//取收集瓶暂存工位到仓库
		80:
			ParameterList3:=2;            //取2号大夹持工具
			A00_取放工具();
			IF 取工具完成 THEN
				取工具完成:=FALSE;
				机器人流程:=81;
			END_IF
		81:
			A71_取暂存收集瓶放仓库();
			IF 取暂存收集瓶组放仓库完成 THEN
				collect_Old_Plate_Slot:=0;
				FunctionID:=0;
				机器人流程:=0;
				取暂存收集瓶组放仓库完成:=FALSE;
			END_IF		
		
		
		
		
		
	
	
	


//取收集器暂存工位到仓库
		90:
			ParameterList3:=2;            //取2号大夹持工具
			A00_取放工具();
			IF 取工具完成 THEN
				取工具完成:=FALSE;
				机器人流程:=91;
			END_IF
		91:
			A70_取暂存收集器组放仓库();
			IF 取暂存收集器组放仓库完成 THEN
				scrape_Old_Plate_Slot:=0;
				FunctionID:=0;
				机器人流程:=0;
				取暂存收集器组放仓库完成:=FALSE;
			END_IF	







//取暂存收集器到刮取位
		100:
			ParameterList3:=3;                           //取3号小夹持工具
			A00_取放工具();
			IF 取工具完成 THEN
				取工具完成:=FALSE;
				机器人流程:=101;
			END_IF	
		101:
			A45_取暂存收集器放刮板位();
			IF 取暂存收集器放刮板位完成 THEN
				scrape_Consume_Slot:=0;
				FunctionID:=0;
				取暂存收集器放刮板位完成:=FALSE;
				机器人流程:=0;
			END_IF
			
			






//取刮板拍照收集器到收集工位
		110:
			ParameterList3:=3;                           //取3号小夹持工具
			A00_取放工具();
			IF 取工具完成 THEN
				取工具完成:=FALSE;
				机器人流程:=111;
			END_IF
		111:
			A55_取刮板收集器放到收集工位();
			IF 取刮板收集器放到收集工位完成 THEN
				FunctionID:=0;
				取刮板收集器放到收集工位完成:=FALSE;
				机器人流程:=0;
			END_IF
			
	
	
	
	
	
	
	
//取暂存收集瓶到收集工位	
		120:
			ParameterList3:=3;                           //取3号小夹持工具
			A00_取放工具();
			IF 取工具完成 THEN
				取工具完成:=FALSE;
				机器人流程:=121;
			END_IF
		121:
			A50_取暂存收集瓶放收集工位();
			IF 取暂存收集瓶放收集工位完成 THEN
				FunctionID:=0;
				取暂存收集瓶放收集工位完成:=FALSE;
				机器人流程:=0;
			END_IF
			
			






//取收集器到暂存工位
		130:
			ParameterList3:=3;                           //取3号小夹持工具
			A00_取放工具();
			IF 取工具完成 THEN
				取工具完成:=FALSE;
				机器人流程:=131;
			END_IF
		131:
			A60_取收集器放暂存工位();
			IF 取收集器放暂存工位完成 THEN
				collect_Powder_Return_Slot:=0;
				收集器组站位符:=FALSE;
				收集工位放收集器完成:=TRUE;
				FunctionID:=0;
				机器人流程:=0;
				取收集器放暂存工位完成:=FALSE;
			END_IF
			
			




//取收集瓶到暂存工位
		140:
			ParameterList3:=3;                           //取3号小夹持工具
			A00_取放工具();
			IF 取工具完成 THEN
				取工具完成:=FALSE;
				机器人流程:=141;
			END_IF
		141:
			A65_取收集瓶放暂存工位();
			IF 取收集瓶放暂存工位完成 THEN
				scrape_Consume_Slot:=0;
				收集瓶组站位符:=FALSE;
				FunctionID:=0;
				机器人流程:=0;
				取收集瓶放暂存工位完成:=FALSE;
			END_IF
			


    END_CASE
END_IF

ACTION A55_取刮板收集器放到收集工位:



CASE 取刮板收集器放到收集工位step OF
	0:
		地轨轴11YDATE.fAbsTarget:=HMI_地轨轴11Y.position[2];     //地轨去取收集组位置暂存位置
			地轨轴11YDATE.xMoveAbs:=TRUE;
			取刮板收集器放到收集工位step:=1;
	1:
		IF 地轨轴11YDATE.bAbMoveDone AND 拍照工位允许取收集器 AND  Status=0 THEN
			地轨轴11YDATE.xMoveAbs:=FALSE;
			拍照工位机器人退出工位完成:=FALSE;
			FunctionID:=11;
			Execute:=1;
			ParameterList5:=4;                          //机器人去夹持工位
			取刮板收集器放到收集工位step:=10;
		END_IF
	10:
		IF RO_ParameterList5=4 THEN
			拍照工位机器人到达收集器夹持位:=TRUE;
			取刮板收集器放到收集工位step:=20;
		END_IF
	20:
		IF 拍照工位机器人退出 THEN
			
			拍照工位机器人到达收集器夹持位:=FALSE;
			ParameterList5:=5;                          //机器人退出工位
			取刮板收集器放到收集工位step:=30;
		END_IF
	30:
		IF RO_ParameterList5=5 THEN
			拍照工位机器人退出完成:=TRUE;
			Execute:=0;
			地轨轴11YDATE.fAbsTarget:=HMI_地轨轴11Y.position[3];     //地轨去收集工位
			地轨轴11YDATE.xMoveAbs:=TRUE;
			取刮板收集器放到收集工位step:=40;
		END_IF
	40:
		IF 地轨轴11YDATE.bAbMoveDone THEN
			地轨轴11YDATE.xMoveAbs:=FALSE;                     
			取刮板收集器放到收集工位step:=50;
		END_IF
	50:
		IF 收集工位允许放收集器 AND  Status=0 THEN
			FunctionID:=12;                             //放收集工位收集器
			ParameterList8:=1;                         //机器人放收集器到夹持工位
			Execute:=1;
			取刮板收集器放到收集工位step:=60;
		END_IF
	60:
		IF RO_ParameterList8=1 THEN
			
			收集工位放收集器到工位:=TRUE;
			取刮板收集器放到收集工位step:=70;
		END_IF
	70:
		IF 收集工位允许机器人退出工位 THEN
			ParameterList8:=2;                     //机器人退出工位
			取刮板收集器放到收集工位step:=80;
		END_IF
	80:
		IF RO_ParameterList8=2 AND Status=2 THEN                //机器人退出工位完成
			Execute:=0;
			收集工位机器人退出完成:=TRUE;
			收集工位放收集器到工位:=FALSE;
			取刮板收集器放到收集工位完成:=TRUE;
			取刮板收集器放到收集工位step:=0;
		END_IF
END_CASE
END_ACTION

ACTION A00_取放工具:



CASE 取工具setp OF
	0:
		IF RO_ParameterList3=ParameterList3 THEN
			取工具完成:=TRUE;
			取工具setp:=0;
		ELSE
			取工具setp:=5;
		END_IF
	5:
		地轨轴11YDATE.fAbsTarget:=HMI_地轨轴11Y.position[4];     //地轨去取工具位置
		地轨轴11YDATE.xMoveAbs:=TRUE;
		IF 地轨轴11YDATE.bAbMoveDone THEN
			地轨轴11YDATE.xMoveAbs:=FALSE;
			FunctionID:=23;                              //取工具ID
			Execute:=1;                                  //机器人启动                        
			取工具setp:=10;
		END_IF
	10:
		IF RO_ParameterList3=ParameterList3 AND Status=2 THEN                               //取工具完成                                   
			Execute:=0;
			取工具完成:=TRUE;
			取工具setp:=0;
		END_IF
END_CASE
END_ACTION

ACTION A15_放点样硅胶板:



CASE 放点样硅胶板step OF
	0:	IF  Status=0 THEN
	  		ParameterList4:=0;
			FunctionID:=2;                         //放点样硅胶板
			ParameterList2:=1;                     //机器人放硅胶板
			Execute:=1;
			放点样硅胶板step:=10;
	  	END_IF
		
	10:
		IF RO_ParameterList2=1 AND Status=2 THEN         //机器人放硅胶板完成
			上样点样放硅胶板完成:=TRUE;
			Execute:=0;
			放点样硅胶板完成:=TRUE;
			放点样硅胶板step:=0;
		END_IF
END_CASE
END_ACTION

ACTION A65_取收集瓶放暂存工位:

CASE 取收集瓶放暂存工位step OF
	0:
		地轨轴11YDATE.fAbsTarget:=HMI_地轨轴11Y.position[3];     //地轨去取收集组位置暂存位置
			地轨轴11YDATE.xMoveAbs:=TRUE;
			取收集瓶放暂存工位step:=5;
	5:
		IF 地轨轴11YDATE.bAbMoveDone AND 收集工位允许机器人取收集瓶放暂存工位 THEN
			地轨轴11YDATE.xMoveAbs:=FALSE;
			收集工位放收集瓶完成:=FALSE;
			FunctionID:=12;
			ParameterList8:=4;                               //到收集工位取收集瓶
			Execute:=1;
			取收集瓶放暂存工位step:=6;
		END_IF
	6:
		
		IF  RO_ParameterList8=4 AND Status=2 THEN
			取收集瓶放暂存工位step:=10;
			收集工位机器人放收集瓶到暂存工位完成:=TRUE;
			Execute:=0;
		END_IF
	10:
		IF Status=0 THEN
			ParameterList8:=5;                               //放收集瓶到暂存工位
			Execute:=1;
			ParameterList9:=collect_Consume_Slot;
			取收集瓶放暂存工位step:=20;
		END_IF
	20:
		IF RO_ParameterList8=5 AND Status=2 THEN                         //放收集瓶到暂存工位完成
			Execute:=0;
			取收集瓶放暂存工位step:=0;
			取收集瓶放暂存工位完成:=TRUE;
		END_IF
END_CASE
END_ACTION

ACTION A71_取暂存收集瓶放仓库:






CASE 取暂存收集瓶组放仓库step OF
	0:
		地轨轴11YDATE.fAbsTarget:=HMI_地轨轴11Y.position[3];     //地轨去取收集组位置暂存位置
		地轨轴11YDATE.xMoveAbs:=TRUE;
		溶液收集瓶定位自动:=FALSE;
		取暂存收集瓶组放仓库step:=10;
	10:
		IF 地轨轴11YDATE.bAbMoveDone AND  Status=0 THEN
			地轨轴11YDATE.xMoveAbs:=FALSE;
			FunctionID:=14;                              //放收集器/瓶到仓库
			ParameterList6:=16;                          //取暂存收集器组
			Execute:=1; 
			取暂存收集瓶组放仓库step:=20;
		END_IF
	20:
		IF RO_ParameterList6=16 AND Status=2 THEN                      //取完成
			Execute:=0; 
			地轨轴11YDATE.fAbsTarget:=HMI_地轨轴11Y.position[6];     //地轨去放收集组位置
			地轨轴11YDATE.xMoveAbs:=TRUE;
			取暂存收集瓶组放仓库step:=30;
		END_IF
	30:
		IF 地轨轴11YDATE.bAbMoveDone AND Status=0 THEN
			地轨轴11YDATE.xMoveAbs:=FALSE;
			ParameterList6:=collect_Old_Plate_Slot+6;               //取暂存收集瓶组
			Execute:=1; 
			取暂存收集瓶组放仓库step:=40;
		END_IF
	40:
		IF RO_ParameterList6=collect_Old_Plate_Slot+6  AND Status=2 THEN
			取暂存收集瓶组放仓库完成:=TRUE;
			Execute:=0; 
			取暂存收集瓶组放仓库step:=0;
		END_IF
END_CASE
END_ACTION

ACTION A20_取点样硅胶板:



CASE 取点样硅胶板step OF
	0:
		地轨轴11YDATE.fAbsTarget:=HMI_地轨轴11Y.position[1];     //地轨去上样点样位置
			地轨轴11YDATE.xMoveAbs:=TRUE;
			IF 地轨轴11YDATE.bAbMoveDone THEN
				地轨轴11YDATE.xMoveAbs:=FALSE; 
				取点样硅胶板step:=5;
			END_IF
	5:
		IF  Status=0 THEN    //上样点样完成，展开准备完成
			FunctionID:=3;                              //取点样硅胶板
			ParameterList2:=2;                          //取硅胶板参数
			Execute:=1;                                  //机器人启动                        
			取点样硅胶板step:=10;
		END_IF
	10:
		IF RO_ParameterList2=2 AND Status=2 THEN
			Execute:=0;
			ParameterList2:=0;
			上样点样允许取硅胶板:=FALSE;
			取点样硅胶板完成:=TRUE;
			取点样硅胶板step:=0;
		END_IF
END_CASE
END_ACTION

ACTION A60_取收集器放暂存工位:


CASE 取收集器放暂存工位step OF
	0:
		地轨轴11YDATE.fAbsTarget:=HMI_地轨轴11Y.position[3];     //地轨去取收集组位置暂存位置
			地轨轴11YDATE.xMoveAbs:=TRUE;
			取收集器放暂存工位step:=5;
			
	5:
		IF 地轨轴11YDATE.bAbMoveDone  THEN
			地轨轴11YDATE.xMoveAbs:=FALSE;
			FunctionID:=12;  
			ParameterList8:=6;                               //放收集器回暂存工位
			Execute:=1;
			取收集器放暂存工位step:=10;
		END_IF
	10:
		IF RO_ParameterList8=6  THEN                       //放收集器回暂存工位完成
			收集工位机器人到达收集器位置:=TRUE;
			取收集器放暂存工位step:=30;
		END_IF
	30:
		IF 收集工位机器人取收集器放回暂存工位 THEN
			ParameterList8:=7;                               //机器人去取收集器
			ParameterList7:=collect_Powder_Return_Slot;
			收集工位机器人取收集器放回暂存工位:=FALSE;
			取收集器放暂存工位step:=40;
		END_IF
	40:
		IF RO_ParameterList8=7 AND Status=2 THEN                         //到达夹持位置
			Execute:=0;
			取收集器放暂存工位完成:=TRUE;
			取收集器放暂存工位step:=0;
		END_IF
END_CASE
END_ACTION

ACTION A10_取升降机硅胶板:


CASE 取升降硅胶板step OF
		0:
			地轨轴11YDATE.fAbsTarget:=HMI_地轨轴11Y.position[1];     //地轨去上样点样位置
			地轨轴11YDATE.xMoveAbs:=TRUE;
			IF 地轨轴11YDATE.bAbMoveDone THEN
				地轨轴11YDATE.xMoveAbs:=FALSE; 
				IF 升降上料伺服允许取料 AND Status=0 THEN
					FunctionID:=1;                              //取升降硅胶板ID
					ParameterList4:=1;                           //去升降机构位置
					Execute:=1;                                  //机器人启动 
					取升降硅胶板step:=10;
				END_IF
			END_IF
			
		10:
			IF RO_ParameterList4=1 THEN                   //机器人到位
				升降上料机器人已吸住物料:=TRUE;
				取升降硅胶板step:=15;
			END_IF
		15:
			IF 升降上料伺服下降完成  THEN
				ParameterList4:=2;                        //机器人取物料
				取升降硅胶板step:=20;
			END_IF
			
		20:
			IF RO_ParameterList4=2 AND Status=2 THEN                //机器人取物料完成
				ParameterList4:=0;
				Execute:=0;
				升降上料机器人取料完成:=TRUE;
				取升降硅胶板完成:=TRUE;
				取升降硅胶板step:=0;
			END_IF
END_CASE
END_ACTION

ACTION A25_放展缸硅胶板:



CASE 放展缸硅胶板step OF
	0:	
		地轨轴11YDATE.fAbsTarget:=HMI_地轨轴11Y.position[5];     //地轨去展开位
		地轨轴11YDATE.xMoveAbs:=TRUE;
		IF 地轨轴11YDATE.bAbMoveDone AND Status=0 THEN
			地轨轴11YDATE.xMoveAbs:=FALSE;
			展开工位机器人到达准备点:=TRUE;
			放展缸硅胶板step:=5;
		END_IF
	5:
		IF 展开工位允许放硅胶板 THEN
			FunctionID:=4;                              //放展缸硅胶板
			Execute:=1;                                  //机器人启动       
			展开工位机器人到达准备点:=FALSE;
			放展缸硅胶板step:=10;
		END_IF
			
	10:
		IF RO_ParameterList1>0 AND Status=2 THEN                       //放硅胶板完成
			展开工位机器人放硅胶板完成:=TRUE;
			FunctionID:=0;
			Execute:=0;
			放展缸硅胶板step:=0;
		END_IF
END_CASE
END_ACTION

ACTION A41_取收集瓶组放暂存工位:


CASE 取收集瓶组放暂存工位step OF
	0:
			地轨轴11YDATE.fAbsTarget:=HMI_地轨轴11Y.position[6];     //地轨去取收集组位置
			地轨轴11YDATE.xMoveAbs:=TRUE;
			溶液收集瓶定位自动:=FALSE;
			取收集瓶组放暂存工位step:=10;
	10:
		IF 地轨轴11YDATE.bAbMoveDone AND Status=0 THEN
				地轨轴11YDATE.xMoveAbs:=FALSE;
				FunctionID:=21;                              //取收集瓶组
				ParameterList6:=collect_Fetch_Rack_Plate+6;       //取收集瓶组坐标
				Execute:=1;                                  //机器人启动                        
				取收集瓶组放暂存工位step:=20;
			END_IF
	20:
		IF RO_ParameterList6=ParameterList6 AND Status=2 THEN             //取收集瓶组完成
			Execute:=0;
			地轨轴11YDATE.fAbsTarget:=HMI_地轨轴11Y.position[3];     //地轨去收集工位
			地轨轴11YDATE.xMoveAbs:=TRUE;
			取收集瓶组放暂存工位step:=30;
		END_IF
	30:
		IF 地轨轴11YDATE.bAbMoveDone AND Status=0 THEN
				地轨轴11YDATE.xMoveAbs:=FALSE;
				FunctionID:=22;                              //放收集瓶组
				ParameterList6:=14;                         //放收集瓶组
				Execute:=1;                                  //机器人启动                        
				取收集瓶组放暂存工位step:=40;
		END_IF
	40:
		IF RO_ParameterList6=14 AND Status=2 THEN                        //放收集瓶完成
			Execute:=0; 
			ParameterList6:=0;
			溶液收集瓶定位自动:=TRUE;
			取收集瓶组放暂存工位完成:=TRUE;
			取收集瓶组放暂存工位step:=0;
		END_IF
END_CASE
END_ACTION

ACTION A65_放废料硅胶板:



CASE 取刮板硅胶板放废料区step OF
	0:
		地轨轴11YDATE.fAbsTarget:=HMI_地轨轴11Y.position[1];     //地轨去上样点样位置
			地轨轴11YDATE.xMoveAbs:=TRUE;
			IF 地轨轴11YDATE.bAbMoveDone THEN
				地轨轴11YDATE.xMoveAbs:=FALSE;
				取刮板硅胶板放废料区step:=5;
            END_IF
	5:
		IF  升降下料伺服允许放料 AND  Status=0 THEN
			
			FunctionID:=8; 
			ParameterList4:=3;                                     //机器人放到废料区
			Execute:=1; 
			取刮板硅胶板放废料区step:=10;
		END_IF
	10:
		IF RO_ParameterList4=3 AND Status=2  THEN                               //机器人放废料区完成
			Execute:=0; 
			刮板拍照工位站位符:=FALSE;
			升降下料机器人放废料完成:=TRUE;
			取刮板硅胶板放废料区完成:=TRUE;
			取刮板硅胶板放废料区step:=0;
		END_IF
END_CASE
END_ACTION

ACTION A35_放拍照硅胶板:




CASE 放拍照硅胶板step OF
	0:
		地轨轴11YDATE.fAbsTarget:=HMI_地轨轴11Y.position[2];     //地轨去刮板拍照位
		地轨轴11YDATE.xMoveAbs:=TRUE;
		IF 地轨轴11YDATE.bAbMoveDone AND Status=0 THEN
				地轨轴11YDATE.xMoveAbs:=FALSE;
				FunctionID:=6;                              //放拍照硅胶板
				ParameterList5:=1;                           //放硅胶板到刮板拍照位
				Execute:=1;                                  //机器人启动                        
				放拍照硅胶板step:=10;
		END_IF
	10:
		IF RO_ParameterList5=1 AND Status=2 THEN              //放硅胶板完成
			Execute:=0; 
			ParameterList5:=0;
			拍照工位放硅胶板完成:=TRUE;
			放拍照硅胶板完成:=TRUE;
			放拍照硅胶板step:=0;
		END_IF
END_CASE
END_ACTION

ACTION A45_取暂存收集器放刮板位:


CASE 取暂存收集器放刮板位step OF
	0:
		IF RO_ParameterList3=3 THEN
			ParameterList3:=0;
			Execute:=0;
			地轨轴11YDATE.fAbsTarget:=HMI_地轨轴11Y.position[2];     //地轨去刮板拍照位
			地轨轴11YDATE.xMoveAbs:=TRUE;
			取暂存收集器放刮板位step:=10;
		END_IF
	10:
		IF 地轨轴11YDATE.bAbMoveDone THEN
			地轨轴11YDATE.xMoveAbs:=FALSE;                     
			取暂存收集器放刮板位step:=20;
		END_IF
	20:
		IF 拍照工位允许放收集器 AND Status=0 THEN
			FunctionID:=9;                              //取暂存收集器
			ParameterList7:=scrape_Consume_Slot;           //取收集器
			Execute:=1;
			取暂存收集器放刮板位step:=30;
		END_IF
	30:
		IF RO_ParameterList7=ParameterList7  THEN                   //取收集器完成
			Execute:=0;
			取暂存收集器放刮板位step:=40;
		END_IF
	40:
		IF Status=0 THEN
			FunctionID:=10;                             //放收集器
			ParameterList5:=2;                         //机器人放收集器到夹持工位
			Execute:=1;
			取暂存收集器放刮板位step:=45;
		END_IF
	45:
		IF RO_ParameterList5=2 THEN
			拍照工位机器人到达夹持位:=TRUE;
			取暂存收集器放刮板位step:=50;
		END_IF
	50:
		IF 拍照工位机器人退出工位 THEN
			ParameterList5:=3;                         //机器人退出工位
			拍照工位机器人到达夹持位:=FALSE;
			取暂存收集器放刮板位step:=60;
		END_IF
	60:
		IF RO_ParameterList5=3 AND Status=2 THEN                    //机器人退出工位完成
			Execute:=0;
			拍照工位机器人退出工位完成:=TRUE;
			取暂存收集器放刮板位完成:=TRUE;
			取暂存收集器放刮板位step:=0;
		END_IF	
	
	
	
	
END_CASE
END_ACTION

ACTION A40_取收集器组放暂存工位:




CASE 取收集器组放暂存工位step OF
	0:
		地轨轴11YDATE.fAbsTarget:=HMI_地轨轴11Y.position[6];     //地轨去取收集组位置
		地轨轴11YDATE.xMoveAbs:=TRUE;
		取收集器组放暂存工位step:=10;
	
	10:
		IF 地轨轴11YDATE.bAbMoveDone  AND Status=0 THEN
				地轨轴11YDATE.xMoveAbs:=FALSE;
				FunctionID:=19;                              //取收集器组
				ParameterList6:=scrape_Fetch_Rack_Plate;       //取收集器组坐标
				Execute:=1;                                  //机器人启动                        
				取收集器组放暂存工位step:=20;
			END_IF
	20:
		IF RO_ParameterList6=ParameterList6 AND Status=2 THEN             //取收集器组完成
			Execute:=0;
			地轨轴11YDATE.fAbsTarget:=HMI_地轨轴11Y.position[3];     //地轨去收集
			地轨轴11YDATE.xMoveAbs:=TRUE;
			取收集器组放暂存工位step:=30;
		END_IF
	30:
		IF 地轨轴11YDATE.bAbMoveDone AND Status=0 THEN
				地轨轴11YDATE.xMoveAbs:=FALSE;
				FunctionID:=20;                              //放收集器组
				ParameterList6:=13;                         //取收集器组坐标
				Execute:=1;                                  //机器人启动                        
				取收集器组放暂存工位step:=40;
		END_IF
	40:
		IF RO_ParameterList6=13  AND Status=2 THEN                        //放收集器完成
			Execute:=0; 
			粉末收集器定位自动:=TRUE;
			取收集器组放暂存工位完成:=TRUE;
			取收集器组放暂存工位step:=0;
		END_IF
	
END_CASE
END_ACTION

ACTION A50_取暂存收集瓶放收集工位:




CASE 取暂存收集瓶放收集工位step OF
	0:
		地轨轴11YDATE.fAbsTarget:=HMI_地轨轴11Y.position[3];     //地轨去取收集组位置暂存位置
			地轨轴11YDATE.xMoveAbs:=TRUE;
			取暂存收集瓶放收集工位step:=1;
	1:
		IF 地轨轴11YDATE.bAbMoveDone AND Status=0 THEN
			地轨轴11YDATE.xMoveAbs:=FALSE;
			FunctionID:=13;                             //取收集瓶
			ParameterList9:=collect_Consume_Slot;           //取收集瓶参数
			Execute:=1;
			取暂存收集瓶放收集工位step:=5;
		END_IF
	5:
		IF RO_ParameterList9=ParameterList9 AND 收集工位允许放收集瓶 THEN        //取收集瓶完成
			Execute:=0;
			取暂存收集瓶放收集工位step:=6;
		END_IF
	6:
		IF Status=0 THEN
			FunctionID:=15;  
			ParameterList8:=3;
			Execute:=1;
			取暂存收集瓶放收集工位step:=10;
		END_IF
	10:
		IF RO_ParameterList8=3 AND Status=2 THEN
				Execute:=0;
			收集工位放收集瓶完成:=TRUE;
			取暂存收集瓶放收集工位完成:=TRUE;
			取暂存收集瓶放收集工位step:=0;
		END_IF
END_CASE
END_ACTION

ACTION A70_取暂存收集器组放仓库:


CASE 取暂存收集器组放仓库step OF
	0:
		IF RO_ParameterList3=2 THEN
			Execute:=0; 
			地轨轴11YDATE.fAbsTarget:=HMI_地轨轴11Y.position[3];     //地轨去取收集组位置暂存位置
			地轨轴11YDATE.xMoveAbs:=TRUE;
			取暂存收集器组放仓库step:=10;
			粉末收集器定位自动:=FALSE;
		END_IF
	10:
		IF 地轨轴11YDATE.bAbMoveDone AND  Status=0 THEN
			地轨轴11YDATE.xMoveAbs:=FALSE;
			粉末收集器定位自动:=FALSE;
			溶液收集瓶定位自动:=FALSE;
			FunctionID:=14;                              //放收集器/瓶到仓库
			ParameterList6:=15;                          //取暂存收集器组
			Execute:=1; 
			取暂存收集器组放仓库step:=20;
		END_IF
	20:
		IF RO_ParameterList6=15 AND  Status=2 THEN                      //取完成
			Execute:=0; 
			地轨轴11YDATE.fAbsTarget:=HMI_地轨轴11Y.position[6];     //地轨去放收集组位置
			地轨轴11YDATE.xMoveAbs:=TRUE;
			取暂存收集器组放仓库step:=30;
		END_IF
	30:
		IF 地轨轴11YDATE.bAbMoveDone AND  Status=0 THEN
			地轨轴11YDATE.xMoveAbs:=FALSE;
			ParameterList6:=scrape_Old_Plate_Slot;               //取暂存收集器组
			Execute:=1;
			取暂存收集器组放仓库step:=40;
		END_IF
	40:
		IF RO_ParameterList6=scrape_Old_Plate_Slot AND Status=2 THEN
			Execute:=0;
			取暂存收集器组放仓库完成:=TRUE;
			取暂存收集器组放仓库step:=0;
		END_IF
	
END_CASE
END_ACTION

ACTION A30_取展缸硅胶板:




CASE 取展缸硅胶板step OF
	0:
		地轨轴11YDATE.fAbsTarget:=HMI_地轨轴11Y.position[5];     //地轨去展开位
		地轨轴11YDATE.xMoveAbs:=TRUE;
		IF 地轨轴11YDATE.bAbMoveDone THEN
			地轨轴11YDATE.xMoveAbs:=FALSE;
			取展缸硅胶板step:=10;
		END_IF
	10:
		IF  ParameterList1>0 AND Status=0 THEN
			FunctionID:=5;                                  //取展缸硅胶板
			Execute:=1;
			取展缸硅胶板step:=20;
		END_IF
	20:
		IF RO_ParameterList1>0 AND Status=2 THEN                       //取硅胶板完成
			Execute:=0;
			取展缸硅胶板完成:=TRUE;
			取展缸硅胶板step:=0;
		END_IF
END_CASE
END_ACTION

ACTION A32_取拍照硅胶板:
CASE 取拍照硅胶完step OF
	0:
		地轨轴11YDATE.fAbsTarget:=HMI_地轨轴11Y.position[2];     //地轨去刮板拍照位
		地轨轴11YDATE.xMoveAbs:=TRUE;
		IF 地轨轴11YDATE.bAbMoveDone THEN
				地轨轴11YDATE.xMoveAbs:=FALSE;
				取拍照硅胶完step:=5;
		END_IF
	5:		
		IF (拍照工位允许取硅胶板去展开 OR 拍照工位允许取硅胶板放废料区) AND Status=0 THEN    
			FunctionID:=6;                              
			ParameterList5:=6;                           //机器人取硅胶板
			Execute:=1;             
			拍照工位允许取硅胶板去展开 := FALSE;
			取拍照硅胶完step:=10;
		END_IF
	10:
		IF RO_ParameterList5=6 AND Status=2 THEN
			Execute:=0;
			ParameterList6:=0;
			取拍照硅胶板完成:=TRUE;
			取拍照硅胶完step:=0;
		IF 拍照工位允许取硅胶板放废料区 THEN
			拍照工位机器人取硅胶板完成 := TRUE;
		END_IF
		END_IF
END_CASE
END_ACTION

END_PROGRAM

// Device/Application/25_FB_功能块/FB_RB_Control
FUNCTION_BLOCK FB_RB_Control
VAR_INPUT
	StartCmd     : BOOL;
StopCmd      : BOOL;
PauseCmd     : BOOL;
Reset:BOOL;
RobotRunning : BOOL;
RobotStopped : BOOL;
RobotPaused  : BOOL;
RobotAlarm   : BOOL;
PowerOn:BOOL;
END_VAR
VAR_OUTPUT
	StartOut     : BOOL;
StopOut      : BOOL;
PauseOut     : BOOL;
ResetOut:BOOL;
StatusRun    : BOOL;
StatusStop   : BOOL;
StatusPause  : BOOL;
StatusAlarm  : BOOL;
PowerOnOut:BOOL;
END_VAR
VAR
	State        : INT := 0;   // 当前状态
END_VAR

(* ================= 报警优先 ================= *)
IF RobotAlarm THEN
    State := 4;
END_IF

CASE State OF

    (* -------- 0：空闲 -------- *)
    0:
        StartOut := FALSE;
        StopOut  := TRUE;
        PauseOut := FALSE;
		ResetOut:=FALSE;
        IF StartCmd AND NOT RobotAlarm THEN
            State := 1;
        END_IF

    (* -------- 1：运行 -------- *)
    1:
		IF NOT PowerOn THEN
			PowerOnOut:=TRUE;
		ELSE
			PowerOnOut:=FALSE;
		END_IF
		IF PowerOn THEN
			StartOut := TRUE;
			StopOut  := FALSE;
			PauseOut := FALSE;
		END_IF
        

        IF StopCmd THEN
            State := 3;
        ELSIF PauseCmd THEN
            State := 2;
        
        END_IF

    (* -------- 2：暂停 -------- *)
    2:
        PauseOut := TRUE;
		StartOut := FALSE ;
        StopOut  := FALSE;
        IF StopCmd THEN
            State := 3;
        ELSIF  StartCmd AND NOT RobotAlarm THEN
            State := 1;
        END_IF

    (* -------- 3：停止 -------- *)
    3:
        StartOut := FALSE;
        StopOut  := TRUE;
        PauseOut := FALSE;

        IF RobotStopped THEN
            State := 0;
        END_IF

    (* -------- 4：报警 -------- *)
    4:
        StartOut := FALSE;
        StopOut  := TRUE;
        PauseOut := FALSE;

        IF  Reset THEN
			ResetOut:=TRUE;
            State := 0;
        END_IF

END_CASE

(* ================= 状态输出 ================= *)
StatusRun   := (State = 1);
StatusPause := (State = 2);
StatusStop  := (State = 0) OR (State = 3);
StatusAlarm := (State = 4);

END_FUNCTION_BLOCK

// Device/Application/40_Man/Develop_TankDrain
PROGRAM Develop_TankDrain
VAR
	i           : INT;      // 循环索引
    anyDraining : BOOL;     // 全局真空泵控制标志
	// 全局真空泵控制标志
	展开step: INT;
	// 全局真空泵控制标志
	TON_3: TON;
	// 全局真空泵控制标志
	TON_4: TON;
	BlowTimer: ARRAY[1..8] OF TON;
	BlowDuration: TIME := t#30s;
END_VAR




A50_Expand_liquid_discharge_排液();

ACTION A50_Expand_liquid_discharge_排液:

// ══════════════════════════════════════════════════════════════
// 排液控制程序（per-tank 并行 FSM，每扫描周期调用）
// ══════════════════════════════════════════════════════════════
// 程序名：PRG_TankDrain
// 文件名：plc_develop_drain.txt
// 职责：监控 Tank_Drain_Enable[1..8]，触发对应缸的 3 阶段排液流程
// 触发条件：Tank_Drain_Enable[i]=TRUE 且 Tank_State[i]=40
// 完成标志：Tank_Drain_Done[i]=TRUE, Tank_State[i]=99
// 复位方式：PC 写 Tank_Drain_Enable[i]=FALSE → 清 Done；
//           PC 写 Tank_State[i]=0 → 释放缸
// ══════════════════════════════════════════════════════════════
// 3 阶段排液时序（工程师已验证）：
//   Phase A — Draining(50)：开排液阀 + 真空泵，等待 DrainDuration
//   Phase B — BlowAir(55) ：追加开吹气阀，等待 BlowDuration
//   Phase C — CylinderRetract(60)：关所有阀 + 气缸退回，等待到位传感器
// ══════════════════════════════════════════════════════════════
// 硬件拓扑：
//   - 每缸有独立排液电磁阀、吹气电磁阀、气缸（伸出/退回）
//   - 真空泵（大真空泵）全局共享，anyDraining 引用计数式控制
//   - 排液气泡传感器按组共享（仅用于监控，不参与控制逻辑）
//   - 支持 8 缸完全并行排液（各缸 FSM 独立推进）
// ══════════════════════════════════════════════════════════════
// Tank_State 状态转换（排液相关）：
//   40 (Developing)      → 50 (Draining)        : Drain_Enable[i] 触发
//   50 (Draining)        → 55 (BlowAir)         : DrainTimer[i].Q
//   55 (BlowAir)         → 60 (CylinderRetract) : BlowTimer[i].Q
//   60 (CylinderRetract) → 99 (Done)            : 气缸到位传感器
//   99 (Done)            → 0  (Idle)            : PC 写 Tank_State=0
//   50/55/60             → 90 (Error)           : 急停
//   注：55/60 为 PLC 内部子状态，PC 只关心 Drain_Done（state 99）
// ══════════════════════════════════════════════════════════════
// 物理 IO 映射表（工程师变量名 → 缸索引）：
//   i=1: 展缸1排液电池阀1自动 / 展缸1吹气电池阀1自动 / 展缸1气缸1自动 / 展缸1气缸1动点
//   i=2: 展缸1排液电池阀2自动 / 展缸1吹气电池阀2自动 / 展缸1气缸2自动 / 展缸1气缸2动点
//   i=3: 展缸1排液电池阀3自动 / 展缸1吹气电池阀3自动 / 展缸1气缸3自动 / 展缸1气缸3动点
//   i=4: 展缸1排液电池阀4自动 / 展缸1吹气电池阀4自动 / 展缸1气缸4自动 / 展缸1气缸4动点
//   i=5: 展缸2排液电池阀1自动 / 展缸2吹气电池阀1自动 / 展缸2气缸1自动 / 展缸2气缸1动点
//   i=6: 展缸2排液电池阀2自动 / 展缸2吹气电池阀2自动 / 展缸2气缸2自动 / 展缸2气缸2动点
//   i=7: 展缸2排液电池阀3自动 / 展缸2吹气电池阀3自动 / 展缸2气缸3自动 / 展缸2气缸3动点
//   i=8: 展缸2排液电池阀4自动 / 展缸2吹气电池阀4自动 / 展缸2气缸4自动 / 展缸2气缸4动点
//   全局: 大真空泵自动
//   监控: 展缸1排液气泡传感器 / 展缸2排液气泡传感器
// ══════════════════════════════════════════════════════════════



// ══ 急停联锁：排液程序响应急停 ══
IF NOT 急停 THEN
    FOR i := 1 TO 8 DO
        // 急停时将所有排液中的缸（50/55/60）标记为 Error
        IF Tank_State[i] = 50 OR Tank_State[i] = 55 OR Tank_State[i] = 60 THEN
            Tank_State[i] := 90;
        END_IF
        // 停止所有定时器
        DrainTimer[i](IN := FALSE, PT := T#0S);
        BlowTimer[i](IN := FALSE, PT := T#0S);
        // 关闭所有排液阀和吹气阀
        CASE i OF
            1: 展缸1排液电池阀1自动 := FALSE; 展缸1吹气电池阀1自动 := FALSE;
            2: 展缸1排液电池阀2自动 := FALSE; 展缸1吹气电池阀2自动 := FALSE;
            3: 展缸1排液电池阀3自动 := FALSE; 展缸1吹气电池阀3自动 := FALSE;
            4: 展缸1排液电池阀4自动 := FALSE; 展缸1吹气电池阀4自动 := FALSE;
            5: 展缸2排液电池阀1自动 := FALSE; 展缸2吹气电池阀1自动 := FALSE;
            6: 展缸2排液电池阀2自动 := FALSE; 展缸2吹气电池阀2自动 := FALSE;
            7: 展缸2排液电池阀3自动 := FALSE; 展缸2吹气电池阀3自动 := FALSE;
            8: 展缸2排液电池阀4自动 := FALSE; 展缸2吹气电池阀4自动 := FALSE;
        END_CASE
    END_FOR
    // 关闭真空泵
    大真空泵站位[0] := FALSE;
    RETURN;
END_IF

// ══ 主循环：逐缸并行处理排液 FSM ══
FOR i := 1 TO 8 DO
 DrainTimer[i](IN := (Tank_State[i] = 50  AND  (i>4 AND 展缸2溶剂废液检测传感器)) OR (Tank_State[i] = 50 AND (i<5 AND 展缸1溶剂废液检测传感器)) , PT := DrainDuration);

 BlowTimer[i](IN := Tank_State[i] = 55, PT := BlowDuration);
 
    // ── 场景 1：PC 撤销 Drain_Enable → 复位 Done 标志（握手完成）──
    IF NOT Tank_Drain_Enable[i] THEN
        Tank_Drain_Done[i] := FALSE;
        DrainTimer[i](IN := FALSE, PT := T#0S);
        BlowTimer[i](IN := FALSE, PT := T#0S);
        // 注意：不主动修改 Tank_State，由 PC 写 0 释放
    // ── 场景 2：Drain_Enable=TRUE，缸处于 Developing(40)，启动排液 Phase A ──
    ELSIF Tank_Drain_Enable[i] AND Tank_State[i] = 40 THEN
        // 开启排液阀
		大真空泵站位[i] := TRUE;
        CASE i OF
            1: 展缸1排液电池阀1自动 := TRUE;
            2: 展缸1排液电池阀2自动 := TRUE;
            3: 展缸1排液电池阀3自动 := TRUE;
            4: 展缸1排液电池阀4自动 := TRUE;
            5: 展缸2排液电池阀1自动 := TRUE;
            6: 展缸2排液电池阀2自动 := TRUE;
            7: 展缸2排液电池阀3自动 := TRUE;
            8: 展缸2排液电池阀4自动 := TRUE;
        END_CASE
        // 推进状态至 Draining
        Tank_State[i] := 50;
    // ── 场景 3：Phase A — Draining(50)，排液阀开 + 真空泵运行，等待排液定时完成 ──
    ELSIF Tank_State[i] = 50 AND (i<5 AND 展缸1溶剂废液检测传感器) THEN
       
        IF DrainTimer[i].Q THEN
            // 排液定时完成，锁定并复位 DrainTimer
            DrainTimer[i](IN := FALSE, PT := T#0S);
            // 开启吹气阀（排液阀保持开启），进入 Phase B
            CASE i OF
                1: 展缸1吹气电池阀1自动 := TRUE;
                2: 展缸1吹气电池阀2自动 := TRUE;
                3: 展缸1吹气电池阀3自动 := TRUE;
                4: 展缸1吹气电池阀4自动 := TRUE;
                
            END_CASE
            Tank_State[i] := 55;
        END_IF
	ELSIF Tank_State[i] = 50  AND  (i>4AND 展缸2溶剂废液检测传感器) THEN
       
        IF DrainTimer[i].Q THEN
            // 排液定时完成，锁定并复位 DrainTimer
            DrainTimer[i](IN := FALSE, PT := T#0S);
            // 开启吹气阀（排液阀保持开启），进入 Phase B
            CASE i OF
                5: 展缸2吹气电池阀1自动 := TRUE;
                6: 展缸2吹气电池阀2自动 := TRUE;
                7: 展缸2吹气电池阀3自动 := TRUE;
                8: 展缸2吹气电池阀4自动 := TRUE;
            END_CASE
            Tank_State[i] := 55;
        END_IF
    // ── 场景 4：Phase B — BlowAir(55)，吹气阀开，等待吹气定时完成 ──
    ELSIF Tank_State[i] = 55 THEN
        大真空泵站位[i] := FALSE;
        IF BlowTimer[i].Q THEN
            // 吹气完成，锁定并复位 BlowTimer
            BlowTimer[i](IN := FALSE, PT := T#0S);
            // 关闭排液阀和吹气阀，启动气缸退回，进入 Phase C
            CASE i OF
                1: 展缸1排液电池阀1自动 := FALSE; 展缸1吹气电池阀1自动 := FALSE; 展缸1气缸1自动 := FALSE;
                2: 展缸1排液电池阀2自动 := FALSE; 展缸1吹气电池阀2自动 := FALSE; 展缸1气缸2自动 := FALSE;
                3: 展缸1排液电池阀3自动 := FALSE; 展缸1吹气电池阀3自动 := FALSE; 展缸1气缸3自动 := FALSE;
                4: 展缸1排液电池阀4自动 := FALSE; 展缸1吹气电池阀4自动 := FALSE; 展缸1气缸4自动 := FALSE;
                5: 展缸2排液电池阀1自动 := FALSE; 展缸2吹气电池阀1自动 := FALSE; 展缸2气缸1自动 := FALSE;
                6: 展缸2排液电池阀2自动 := FALSE; 展缸2吹气电池阀2自动 := FALSE; 展缸2气缸2自动 := FALSE;
                7: 展缸2排液电池阀3自动 := FALSE; 展缸2吹气电池阀3自动 := FALSE; 展缸2气缸3自动 := FALSE;
                8: 展缸2排液电池阀4自动 := FALSE; 展缸2吹气电池阀4自动 := FALSE; 展缸2气缸4自动 := FALSE;
            END_CASE
            Tank_State[i] := 60;
       END_IF
    // ── 场景 5：Phase C — CylinderRetract(60)，等待气缸退回到位 ──
    ELSIF Tank_State[i] = 60 THEN
        CASE i OF
            1: IF 展缸1气缸1原点 THEN   Tank_State[1] := 65; END_IF
            2: IF 展缸1气缸2原点 THEN   Tank_State[2] := 65; END_IF
            3: IF 展缸1气缸3原点 THEN   Tank_State[3] := 65; END_IF
            4: IF 展缸1气缸4原点 THEN   Tank_State[4] := 65; END_IF
            5: IF 展缸2气缸1原点 THEN   Tank_State[5] := 65; END_IF
            6: IF 展缸2气缸2原点 THEN   Tank_State[6] := 65; END_IF
            7: IF 展缸2气缸3原点 THEN   Tank_State[7] := 65; END_IF
            8: IF 展缸2气缸4原点 THEN   Tank_State[8] := 65; END_IF
        END_CASE
   
	 //场景 6：Phase D — RobotPickup(65)，等待机器人取板（电平握手，串行）──
    ELSIF Tank_State[i] = 65 THEN
		bParameterList1[i]:=TRUE;   //机器人参数取展缸位置
		
        IF RO_ParameterList1=i THEN
            // 机器人空闲 → 发出取板请求（电平保持）
			Tank_State[RO_ParameterList1] := 99;
			bParameterList1[i]:=FALSE;
			CASE i OF
            1:  Tank_Drain_Done[1] := TRUE; 
            2:   Tank_Drain_Done[2] := TRUE; 
            3:   Tank_Drain_Done[3] := TRUE;  
            4:   Tank_Drain_Done[4] := TRUE;  
            5:   Tank_Drain_Done[5] := TRUE;  
            6:   Tank_Drain_Done[6] := TRUE;  
            7:   Tank_Drain_Done[7] := TRUE;  
            8:   Tank_Drain_Done[8] := TRUE;  
        END_CASE
//             RobotRequested := TRUE;
//             Robot_Pickup_Req := TRUE;
//             Robot_Source_Tank := i;
        END_IF
//         IF RobotRequested AND Robot_Source_Tank = i AND Robot_Pickup_Done THEN
//             // 机器人取板完成 → 清除握手信号，标记排液完成
//             Robot_Pickup_Req := FALSE;
//             RobotRequested := FALSE;
//             Tank_Drain_Done[i] := TRUE;
//             
//         END_IF
	END_IF
	

END_FOR

// ══ 真空泵全局控制：当无任何缸在排液/吹气时关闭真空泵 ══

IF bParameterList1[1] OR bParameterList1[2]  OR  bParameterList1[3] OR bParameterList1[4] OR bParameterList1[5] OR bParameterList1[6] OR bParameterList1[7] OR bParameterList1[8]THEN
	展开工位允许取硅胶板:=TRUE;
END_IF
IF  展开工位允许取硅胶板 THEN
	IF bParameterList1[1] THEN
		ParameterList1:=1;
	ELSIF bParameterList1[2] THEN
		ParameterList1:=2;
	ELSIF bParameterList1[3] THEN
		ParameterList1:=3;
	ELSIF bParameterList1[4] THEN
		ParameterList1:=4;
	ELSIF bParameterList1[5] THEN
		ParameterList1:=5;
	ELSIF bParameterList1[6] THEN
		ParameterList1:=6;
	ELSIF bParameterList1[7] THEN
		ParameterList1:=7;
	ELSIF bParameterList1[8] THEN
		ParameterList1:=8;
	END_IF
END_IF
END_ACTION

END_PROGRAM

// Device/Application/25_FB_功能块/FB_Mode
FUNCTION_BLOCK FB_Mode
VAR_INPUT
    xStart      : BOOL;  // 启动按钮
    xStop       : BOOL;  // 停止按钮
    xReset      : BOOL;  // 复位按钮
    xAutoMode   : BOOL;  // TRUE=自动模式，FALSE=手动模式
    xFault      : BOOL;  // 故障信号
    xEmergency  : BOOL;  // 急停信号（急停按下为FALSE）
END_VAR
VAR_OUTPUT
    bRed        : BOOL;  // 红灯
    bYellow     : BOOL;  // 黄灯
    bGreen      : BOOL;  // 绿灯
    bBuzzer     : BOOL;  // 蜂鸣器
    iState      : INT;   // 设备状态: 0=停止, 1=运行, 2=故障, 3=急停
    bAuto       : BOOL;  // 自动模式指示
END_VAR
VAR
    iDeviceState : INT := 0;  // 0=停止, 1=运行, 2=故障, 3=急停
    
    // 定时器
    tBuzzerPulse : TON;  // 蜂鸣器脉冲
    tFlashTimer  : TON;  // 闪烁定时器
    tShortBeep   : TON;  // 短鸣定时器
    tEmergencyBeep : TON; // 急停蜂鸣器定时器
	// 蜂鸣器激活
	tEmergencyBeep1: TON;
    
    // 标志
    bBuzzerActive : BOOL := FALSE;  // 蜂鸣器激活
    bFlashFlag    : BOOL;           // 闪烁标志
    bBeepOnce     : BOOL := FALSE;  // 单次蜂鸣标志
    bEmergencyBuzzer : BOOL := FALSE; // 急停蜂鸣器标志
    bEmergencyActive : BOOL := FALSE; // 急停激活标志
	ALT_0: ALT;
	ALT_1: ALT;
	TON_0: TON;
	ALT_2: ALT;
	TON_1: TON;
	TON_2: TON;
END_VAR
VAR_INPUT
	bWarning_alarm: BOOL;
END_VAR

// 模式状态
bAuto := xAutoMode;

// 状态机
CASE iDeviceState OF
    EN_功能块状态.停止:  // 停止状态
        IF NOT xEmergency THEN
            iDeviceState := EN_功能块状态.急停;  // 急停
            bEmergencyActive := TRUE;
        ELSIF xFault THEN
            iDeviceState := EN_功能块状态.故障;  // 故障
            bBuzzerActive := TRUE;
        ELSIF (bAuto AND xStart)  THEN
		 bBeepOnce := TRUE;  // 启动短鸣
		  iDeviceState := EN_功能块状态.初始化;  // 初始化

        END_IF;
    
    EN_功能块状态.运行:  // 运行状态
        IF NOT xEmergency THEN
            iDeviceState := EN_功能块状态.急停;  // 急停
            bEmergencyActive := TRUE;
        ELSIF xFault THEN
            iDeviceState := EN_功能块状态.故障;  // 故障
            bBuzzerActive := TRUE;
        ELSIF xStop THEN
            iDeviceState := EN_功能块状态.停止;  // 停止
            bBeepOnce := TRUE;  // 停止短鸣
        END_IF;
        
    EN_功能块状态.故障:  // 故障状态
        IF NOT xEmergency THEN
            iDeviceState := EN_功能块状态.急停;  // 急停
            bEmergencyActive := TRUE;
        ELSIF xReset AND NOT xFault THEN
            iDeviceState := EN_功能块状态.停止;  // 停止
            bBuzzerActive := FALSE;
			bBuzzer:=FALSE;
        END_IF;
        
    EN_功能块状态.急停:  // 急停状态
        // 急停复位需要：急停信号解除 + 复位按钮按下
        IF  xEmergency AND xReset THEN
            iDeviceState := EN_功能块状态.停止;  // 停止
            bEmergencyActive := FALSE;
            bEmergencyBuzzer := FALSE;
			bBuzzer:=FALSE;
        END_IF;
	EN_功能块状态.初始化:  //初始化状态
	 TON_0(IN:=TRUE , PT:=T#3S );
		IF TON_0.Q THEN
		iDeviceState := EN_功能块状态.运行;  // 运行
		END_IF 
END_CASE;

// 急停蜂鸣器控制（急停时蜂鸣器以不同频率鸣响）
IF  bEmergencyActive THEN
    tEmergencyBeep(IN := NOT tEmergencyBeep.Q, PT := T#2S );
	ALT_1(xExecute:= tEmergencyBeep.Q, xOut:=bBuzzer );  // 急停时蜂鸣器响2秒，停2秒	
END_IF;

//三色灯控制
// 闪烁定时器
tFlashTimer(IN := NOT tFlashTimer.Q, PT := T#500MS);
ALT_0(xExecute:=tFlashTimer.Q , xOut:=bFlashFlag );

CASE iDeviceState OF
    EN_功能块状态.停止:  // 停止状态
        IF bAuto THEN
            bYellow := TRUE;           // 自动模式：黄灯常亮
        ELSE
            bYellow := bFlashFlag;     // 手动模式：黄灯闪烁
        END_IF;
		 bGreen :=FALSE;
		 bRed :=FALSE;
        
    EN_功能块状态.运行:  // 运行状态
        bGreen := TRUE;
         bRed :=FALSE;
		  bYellow := FALSE; 
    EN_功能块状态.故障:  // 故障状态
        bRed := TRUE;
         bGreen :=FALSE;
		 bYellow := FALSE; 
    EN_功能块状态.急停:  // 急停状态
        bRed := bFlashFlag;  // 红灯闪烁
		bGreen :=FALSE;
		 bYellow := FALSE; 
END_CASE;
tShortBeep(IN := bBeepOnce AND NOT bEmergencyActive, PT := T#500MS);
// 蜂鸣器控制
IF bBeepOnce AND NOT bEmergencyActive THEN
	bBuzzer := TRUE;  // 短鸣
    IF tShortBeep.Q THEN
        bBeepOnce := FALSE;
       bBuzzer := FALSE;
    END_IF;
    
END_IF;

// 故障时蜂鸣器（非急停状态时生效）
IF NOT bEmergencyActive AND xFault  THEN
    tBuzzerPulse(IN := NOT tBuzzerPulse.Q, PT := T#500MS);
ALT_2(xExecute:= tBuzzerPulse.Q, xOut:= bBuzzer);
END_IF;


//蜂鸣器5S后停止
TON_2(IN:=iDeviceState=2 OR iDeviceState=3 OR bWarning_alarm ,PT:=T#5S);
IF TON_2.Q THEN
	bBuzzer:=FALSE;
END_IF

IF bWarning_alarm AND NOT TON_2.Q THEN
	bBuzzer:=TRUE;
	
END_IF
IF bWarning_alarm  THEN
	 bRed := TRUE;
	  
END_IF

IF xReset THEN
	bBuzzer:=FALSE;
	bRed := FALSE;
END_IF



// 输出状态
iState := iDeviceState;

END_FUNCTION_BLOCK

// Device/Application/40_Man/initialization
PROGRAM initialization
VAR
END_VAR

上样轴4X轴DATE.bHomed:=FALSE;
上样轴5Z轴DATE.bHomed:=FALSE;

END_PROGRAM

(* text CNC_2
N0 E200 E-200
N1 F5000


N00050 G1 X200 Y20
N00051 G1 X100 Y0
N052 G01 X0150 Y30 
N00911 G1 X335 Y0
*)

(* text CNC_1
N0 E200 E-200
N1 F5000
N2 G53
N00040 G0 Z 5.0F500
N00050 G0 X$g_sx[1]$ Y$g_sy[1]$
N00060 G0 Z $g_pass_z$F500
N00061 M10
N00090 G1 X$g_sx[1]$ Y$g_sy[1]$ F$g_scrape_feed$
N00100 G1 X$g_sx[2]$ Y$g_sy[2]$ F$g_scrape_feed$
N00110 G1 X$g_sx[3]$ Y$g_sy[3]$ F$g_scrape_feed$
N00120 G1 X$g_sx[4]$ Y$g_sy[4]$ F$g_scrape_feed$
N00130 G1 X$g_sx[5]$ Y$g_sy[5]$ F$g_scrape_feed$
N00140 G1 X$g_sx[6]$ Y$g_sy[6]$ F$g_scrape_feed$
N00150 G1 X$g_sx[7]$ Y$g_sy[7]$ F$g_scrape_feed$
N00160 G1 X$g_sx[8]$ Y$g_sy[8]$ F$g_scrape_feed$
N00170 G1 X$g_sx[9]$ Y$g_sy[9]$ F$g_scrape_feed$
N00180 G1 X$g_sx[10]$ Y$g_sy[10]$ F$g_scrape_feed$
N00190 G1 X$g_sx[11]$ Y$g_sy[11]$ F$g_scrape_feed$
N00200 G1 X$g_sx[12]$ Y$g_sy[12]$ F$g_scrape_feed$
N00210 G1 X$g_sx[13]$ Y$g_sy[13]$ F$g_scrape_feed$
N00220 G1 X$g_sx[14]$ Y$g_sy[14]$ F$g_scrape_feed$
N00230 G1 X$g_sx[15]$ Y$g_sy[15]$ F$g_scrape_feed$
N00240 G1 X$g_sx[16]$ Y$g_sy[16]$ F$g_scrape_feed$
N00250 G1 X$g_sx[17]$ Y$g_sy[17]$ F$g_scrape_feed$
N00260 G1 X$g_sx[18]$ Y$g_sy[18]$ F$g_scrape_feed$
N00270 G1 X$g_sx[19]$ Y$g_sy[19]$ F$g_scrape_feed$
N00280 G1 X$g_sx[20]$ Y$g_sy[20]$ F$g_scrape_feed$
N00290 G1 X$g_sx[21]$ Y$g_sy[21]$ F$g_scrape_feed$
N00300 G1 X$g_sx[22]$ Y$g_sy[22]$ F$g_scrape_feed$
N00310 G1 X$g_sx[23]$ Y$g_sy[23]$ F$g_scrape_feed$
N00320 G1 X$g_sx[24]$ Y$g_sy[24]$ F$g_scrape_feed$
N00330 G1 X$g_sx[25]$ Y$g_sy[25]$ F$g_scrape_feed$
N00340 G1 X$g_sx[26]$ Y$g_sy[26]$ F$g_scrape_feed$
N00350 G1 X$g_sx[27]$ Y$g_sy[27]$ F$g_scrape_feed$
N00360 G1 X$g_sx[28]$ Y$g_sy[28]$ F$g_scrape_feed$
N00370 G1 X$g_sx[29]$ Y$g_sy[29]$ F$g_scrape_feed$
N00380 G1 X$g_sx[30]$ Y$g_sy[30]$ F$g_scrape_feed$
N00390 G1 X$g_sx[31]$ Y$g_sy[31]$ F$g_scrape_feed$
N00400 G1 X$g_sx[32]$ Y$g_sy[32]$ F$g_scrape_feed$
N00410 G1 X$g_sx[33]$ Y$g_sy[33]$ F$g_scrape_feed$
N00420 G1 X$g_sx[34]$ Y$g_sy[34]$ F$g_scrape_feed$
N00430 G1 X$g_sx[35]$ Y$g_sy[35]$ F$g_scrape_feed$
N00440 G1 X$g_sx[36]$ Y$g_sy[36]$ F$g_scrape_feed$
N00450 G1 X$g_sx[37]$ Y$g_sy[37]$ F$g_scrape_feed$
N00460 G1 X$g_sx[38]$ Y$g_sy[38]$ F$g_scrape_feed$
N00470 G1 X$g_sx[39]$ Y$g_sy[39]$ F$g_scrape_feed$
N00480 G1 X$g_sx[40]$ Y$g_sy[40]$ F$g_scrape_feed$
N00490 G1 X$g_sx[41]$ Y$g_sy[41]$ F$g_scrape_feed$
N00500 G1 X$g_sx[42]$ Y$g_sy[42]$ F$g_scrape_feed$
N00510 G1 X$g_sx[43]$ Y$g_sy[43]$ F$g_scrape_feed$
N00520 G1 X$g_sx[44]$ Y$g_sy[44]$ F$g_scrape_feed$
N00530 G1 X$g_sx[45]$ Y$g_sy[45]$ F$g_scrape_feed$
N00540 G1 X$g_sx[46]$ Y$g_sy[46]$ F$g_scrape_feed$
N00550 G1 X$g_sx[47]$ Y$g_sy[47]$ F$g_scrape_feed$
N00560 G1 X$g_sx[48]$ Y$g_sy[48]$ F$g_scrape_feed$
N00570 G1 X$g_sx[49]$ Y$g_sy[49]$ F$g_scrape_feed$
N00580 G1 X$g_sx[50]$ Y$g_sy[50]$ F$g_scrape_feed$
N00590 G1 X$g_sx[51]$ Y$g_sy[51]$ F$g_scrape_feed$
N00600 G1 X$g_sx[52]$ Y$g_sy[52]$ F$g_scrape_feed$
N00610 G1 X$g_sx[53]$ Y$g_sy[53]$ F$g_scrape_feed$
N00620 G1 X$g_sx[54]$ Y$g_sy[54]$ F$g_scrape_feed$
N00630 G1 X$g_sx[55]$ Y$g_sy[55]$ F$g_scrape_feed$
N00640 G1 X$g_sx[56]$ Y$g_sy[56]$ F$g_scrape_feed$
N00650 G1 X$g_sx[57]$ Y$g_sy[57]$ F$g_scrape_feed$
N00660 G1 X$g_sx[58]$ Y$g_sy[58]$ F$g_scrape_feed$
N00670 G1 X$g_sx[59]$ Y$g_sy[59]$ F$g_scrape_feed$
N00680 G1 X$g_sx[60]$ Y$g_sy[60]$ F$g_scrape_feed$
N00690 G1 X$g_sx[61]$ Y$g_sy[61]$ F$g_scrape_feed$
N00700 G1 X$g_sx[62]$ Y$g_sy[62]$ F$g_scrape_feed$
N00710 G1 X$g_sx[63]$ Y$g_sy[63]$ F$g_scrape_feed$
N00720 G1 X$g_sx[64]$ Y$g_sy[64]$ F$g_scrape_feed$
N00730 G1 X$g_sx[65]$ Y$g_sy[65]$ F$g_scrape_feed$
N00740 G1 X$g_sx[66]$ Y$g_sy[66]$ F$g_scrape_feed$
N00750 G1 X$g_sx[67]$ Y$g_sy[67]$ F$g_scrape_feed$
N00760 G1 X$g_sx[68]$ Y$g_sy[68]$ F$g_scrape_feed$
N00770 G1 X$g_sx[69]$ Y$g_sy[69]$ F$g_scrape_feed$
N00780 G1 X$g_sx[70]$ Y$g_sy[70]$ F$g_scrape_feed$
N00790 G1 X$g_sx[71]$ Y$g_sy[71]$ F$g_scrape_feed$
N00800 G1 X$g_sx[72]$ Y$g_sy[72]$ F$g_scrape_feed$
N00810 G1 X$g_sx[73]$ Y$g_sy[73]$ F$g_scrape_feed$
N00820 G1 X$g_sx[74]$ Y$g_sy[74]$ F$g_scrape_feed$
N00830 G1 X$g_sx[75]$ Y$g_sy[75]$ F$g_scrape_feed$
N00840 G1 X$g_sx[76]$ Y$g_sy[76]$ F$g_scrape_feed$
N00850 G1 X$g_sx[77]$ Y$g_sy[77]$ F$g_scrape_feed$
N00860 G1 X$g_sx[78]$ Y$g_sy[78]$ F$g_scrape_feed$
N00870 G1 X$g_sx[79]$ Y$g_sy[79]$ F$g_scrape_feed$
N00880 G1 X$g_sx[80]$ Y$g_sy[80]$ F$g_scrape_feed$
N00890 G1 X$g_sx[81]$ Y$g_sy[81]$ F$g_scrape_feed$
N00900 G1 X$g_sx[82]$ Y$g_sy[82]$ F$g_scrape_feed$
N00910 G1 X$g_sx[83]$ Y$g_sy[83]$ F$g_scrape_feed$
N00920 G1 X$g_sx[84]$ Y$g_sy[84]$ F$g_scrape_feed$
N00930 G1 X$g_sx[85]$ Y$g_sy[85]$ F$g_scrape_feed$
N00940 G1 X$g_sx[86]$ Y$g_sy[86]$ F$g_scrape_feed$
N00950 G1 X$g_sx[87]$ Y$g_sy[87]$ F$g_scrape_feed$
N00960 G1 X$g_sx[88]$ Y$g_sy[88]$ F$g_scrape_feed$
N00970 G1 X$g_sx[89]$ Y$g_sy[89]$ F$g_scrape_feed$
N00980 G1 X$g_sx[90]$ Y$g_sy[90]$ F$g_scrape_feed$
N00990 G1 X$g_sx[91]$ Y$g_sy[91]$ F$g_scrape_feed$
N01000 G1 X$g_sx[92]$ Y$g_sy[92]$ F$g_scrape_feed$
N01010 G1 X$g_sx[93]$ Y$g_sy[93]$ F$g_scrape_feed$
N01020 G1 X$g_sx[94]$ Y$g_sy[94]$ F$g_scrape_feed$
N01030 G1 X$g_sx[95]$ Y$g_sy[95]$ F$g_scrape_feed$
N01040 G1 X$g_sx[96]$ Y$g_sy[96]$ F$g_scrape_feed$
N01050 G1 X$g_sx[97]$ Y$g_sy[97]$ F$g_scrape_feed$
N01060 G1 X$g_sx[98]$ Y$g_sy[98]$ F$g_scrape_feed$
N01070 G1 X$g_sx[99]$ Y$g_sy[99]$ F$g_scrape_feed$
N01080 G1 X$g_sx[100]$ Y$g_sy[100]$ F$g_scrape_feed$
N01090 G1 X$g_sx[101]$ Y$g_sy[101]$ F$g_scrape_feed$
N01100 G1 X$g_sx[102]$ Y$g_sy[102]$ F$g_scrape_feed$
N01110 G1 X$g_sx[103]$ Y$g_sy[103]$ F$g_scrape_feed$
N01120 G1 X$g_sx[104]$ Y$g_sy[104]$ F$g_scrape_feed$
N01130 G1 X$g_sx[105]$ Y$g_sy[105]$ F$g_scrape_feed$
N01140 G1 X$g_sx[106]$ Y$g_sy[106]$ F$g_scrape_feed$
N01150 G1 X$g_sx[107]$ Y$g_sy[107]$ F$g_scrape_feed$
N01160 G1 X$g_sx[108]$ Y$g_sy[108]$ F$g_scrape_feed$
N01170 G1 X$g_sx[109]$ Y$g_sy[109]$ F$g_scrape_feed$
N01180 G1 X$g_sx[110]$ Y$g_sy[110]$ F$g_scrape_feed$
N01190 G1 X$g_sx[111]$ Y$g_sy[111]$ F$g_scrape_feed$
N01200 G1 X$g_sx[112]$ Y$g_sy[112]$ F$g_scrape_feed$
N01210 G1 X$g_sx[113]$ Y$g_sy[113]$ F$g_scrape_feed$
N01220 G1 X$g_sx[114]$ Y$g_sy[114]$ F$g_scrape_feed$
N01230 G1 X$g_sx[115]$ Y$g_sy[115]$ F$g_scrape_feed$
N01240 G1 X$g_sx[116]$ Y$g_sy[116]$ F$g_scrape_feed$
N01250 G1 X$g_sx[117]$ Y$g_sy[117]$ F$g_scrape_feed$
N01260 G1 X$g_sx[118]$ Y$g_sy[118]$ F$g_scrape_feed$
N01270 G1 X$g_sx[119]$ Y$g_sy[119]$ F$g_scrape_feed$
N01280 G1 X$g_sx[120]$ Y$g_sy[120]$ F$g_scrape_feed$
N01290 G1 X$g_sx[121]$ Y$g_sy[121]$ F$g_scrape_feed$
N01300 G1 X$g_sx[122]$ Y$g_sy[122]$ F$g_scrape_feed$
N01310 G1 X$g_sx[123]$ Y$g_sy[123]$ F$g_scrape_feed$
N01320 G1 X$g_sx[124]$ Y$g_sy[124]$ F$g_scrape_feed$
N01330 G1 X$g_sx[125]$ Y$g_sy[125]$ F$g_scrape_feed$
N01340 G1 X$g_sx[126]$ Y$g_sy[126]$ F$g_scrape_feed$
N01350 G1 X$g_sx[127]$ Y$g_sy[127]$ F$g_scrape_feed$
N01360 G1 X$g_sx[128]$ Y$g_sy[128]$ F$g_scrape_feed$
N01370 G1 X$g_sx[129]$ Y$g_sy[129]$ F$g_scrape_feed$
N01380 G1 X$g_sx[130]$ Y$g_sy[130]$ F$g_scrape_feed$
N01390 G1 X$g_sx[131]$ Y$g_sy[131]$ F$g_scrape_feed$
N01400 G1 X$g_sx[132]$ Y$g_sy[132]$ F$g_scrape_feed$
N01410 G1 X$g_sx[133]$ Y$g_sy[133]$ F$g_scrape_feed$
N01420 G1 X$g_sx[134]$ Y$g_sy[134]$ F$g_scrape_feed$
N01430 G1 X$g_sx[135]$ Y$g_sy[135]$ F$g_scrape_feed$
N01440 G1 X$g_sx[136]$ Y$g_sy[136]$ F$g_scrape_feed$
N01450 G1 X$g_sx[137]$ Y$g_sy[137]$ F$g_scrape_feed$
N01460 G1 X$g_sx[138]$ Y$g_sy[138]$ F$g_scrape_feed$
N01470 G1 X$g_sx[139]$ Y$g_sy[139]$ F$g_scrape_feed$
N01480 G1 X$g_sx[140]$ Y$g_sy[140]$ F$g_scrape_feed$
N01490 G1 X$g_sx[141]$ Y$g_sy[141]$ F$g_scrape_feed$
N01500 G1 X$g_sx[142]$ Y$g_sy[142]$ F$g_scrape_feed$
N01510 G1 X$g_sx[143]$ Y$g_sy[143]$ F$g_scrape_feed$
N01520 G1 X$g_sx[144]$ Y$g_sy[144]$ F$g_scrape_feed$
N01530 G1 X$g_sx[145]$ Y$g_sy[145]$ F$g_scrape_feed$
N01540 G1 X$g_sx[146]$ Y$g_sy[146]$ F$g_scrape_feed$
N01550 G1 X$g_sx[147]$ Y$g_sy[147]$ F$g_scrape_feed$
N01560 G1 X$g_sx[148]$ Y$g_sy[148]$ F$g_scrape_feed$
N01570 G1 X$g_sx[149]$ Y$g_sy[149]$ F$g_scrape_feed$
N01580 G1 X$g_sx[150]$ Y$g_sy[150]$ F$g_scrape_feed$
N01590 G1 X$g_sx[151]$ Y$g_sy[151]$ F$g_scrape_feed$
N01600 G1 X$g_sx[152]$ Y$g_sy[152]$ F$g_scrape_feed$
N01610 G1 X$g_sx[153]$ Y$g_sy[153]$ F$g_scrape_feed$
N01620 G1 X$g_sx[154]$ Y$g_sy[154]$ F$g_scrape_feed$
N01630 G1 X$g_sx[155]$ Y$g_sy[155]$ F$g_scrape_feed$
N01640 G1 X$g_sx[156]$ Y$g_sy[156]$ F$g_scrape_feed$
N01650 G1 X$g_sx[157]$ Y$g_sy[157]$ F$g_scrape_feed$
N01660 G1 X$g_sx[158]$ Y$g_sy[158]$ F$g_scrape_feed$
N01670 G1 X$g_sx[159]$ Y$g_sy[159]$ F$g_scrape_feed$
N01680 G1 X$g_sx[160]$ Y$g_sy[160]$ F$g_scrape_feed$
N01690 G1 X$g_sx[161]$ Y$g_sy[161]$ F$g_scrape_feed$
N01700 G1 X$g_sx[162]$ Y$g_sy[162]$ F$g_scrape_feed$
N01710 G1 X$g_sx[163]$ Y$g_sy[163]$ F$g_scrape_feed$
N01720 G1 X$g_sx[164]$ Y$g_sy[164]$ F$g_scrape_feed$
N01730 G1 X$g_sx[165]$ Y$g_sy[165]$ F$g_scrape_feed$
N01740 G1 X$g_sx[166]$ Y$g_sy[166]$ F$g_scrape_feed$
N01750 G1 X$g_sx[167]$ Y$g_sy[167]$ F$g_scrape_feed$
N01760 G1 X$g_sx[168]$ Y$g_sy[168]$ F$g_scrape_feed$
N01770 G1 X$g_sx[169]$ Y$g_sy[169]$ F$g_scrape_feed$
N01780 G1 X$g_sx[170]$ Y$g_sy[170]$ F$g_scrape_feed$
N01790 G1 X$g_sx[171]$ Y$g_sy[171]$ F$g_scrape_feed$
N01800 G1 X$g_sx[172]$ Y$g_sy[172]$ F$g_scrape_feed$
N01810 G1 X$g_sx[173]$ Y$g_sy[173]$ F$g_scrape_feed$
N01820 G1 X$g_sx[174]$ Y$g_sy[174]$ F$g_scrape_feed$
N01830 G1 X$g_sx[175]$ Y$g_sy[175]$ F$g_scrape_feed$
N01840 G1 X$g_sx[176]$ Y$g_sy[176]$ F$g_scrape_feed$
N01850 G1 X$g_sx[177]$ Y$g_sy[177]$ F$g_scrape_feed$
N01860 G1 X$g_sx[178]$ Y$g_sy[178]$ F$g_scrape_feed$
N01870 G1 X$g_sx[179]$ Y$g_sy[179]$ F$g_scrape_feed$
N01880 G1 X$g_sx[180]$ Y$g_sy[180]$ F$g_scrape_feed$
N01890 G1 X$g_sx[181]$ Y$g_sy[181]$ F$g_scrape_feed$
N01900 G1 X$g_sx[182]$ Y$g_sy[182]$ F$g_scrape_feed$
N01910 G1 X$g_sx[183]$ Y$g_sy[183]$ F$g_scrape_feed$
N01920 G1 X$g_sx[184]$ Y$g_sy[184]$ F$g_scrape_feed$
N01930 G1 X$g_sx[185]$ Y$g_sy[185]$ F$g_scrape_feed$
N01940 G1 X$g_sx[186]$ Y$g_sy[186]$ F$g_scrape_feed$
N01950 G1 X$g_sx[187]$ Y$g_sy[187]$ F$g_scrape_feed$
N01960 G1 X$g_sx[188]$ Y$g_sy[188]$ F$g_scrape_feed$
N01970 G1 X$g_sx[189]$ Y$g_sy[189]$ F$g_scrape_feed$
N01980 G1 X$g_sx[190]$ Y$g_sy[190]$ F$g_scrape_feed$
N01990 G1 X$g_sx[191]$ Y$g_sy[191]$ F$g_scrape_feed$
N02000 G1 X$g_sx[192]$ Y$g_sy[192]$ F$g_scrape_feed$
N02010 G1 X$g_sx[193]$ Y$g_sy[193]$ F$g_scrape_feed$
N02020 G1 X$g_sx[194]$ Y$g_sy[194]$ F$g_scrape_feed$
N02030 G1 X$g_sx[195]$ Y$g_sy[195]$ F$g_scrape_feed$
N02040 G1 X$g_sx[196]$ Y$g_sy[196]$ F$g_scrape_feed$
N02050 G1 X$g_sx[197]$ Y$g_sy[197]$ F$g_scrape_feed$
N02060 G1 X$g_sx[198]$ Y$g_sy[198]$ F$g_scrape_feed$
N02070 G1 X$g_sx[199]$ Y$g_sy[199]$ F$g_scrape_feed$
N02080 G1 X$g_sx[200]$ Y$g_sy[200]$ F$g_scrape_feed$
N02090 G1 X$g_sx[201]$ Y$g_sy[201]$ F$g_scrape_feed$
N02100 G1 X$g_sx[202]$ Y$g_sy[202]$ F$g_scrape_feed$
N02110 G1 X$g_sx[203]$ Y$g_sy[203]$ F$g_scrape_feed$
N02120 G1 X$g_sx[204]$ Y$g_sy[204]$ F$g_scrape_feed$
N02130 G1 X$g_sx[205]$ Y$g_sy[205]$ F$g_scrape_feed$
N02140 G1 X$g_sx[206]$ Y$g_sy[206]$ F$g_scrape_feed$
N02150 G1 X$g_sx[207]$ Y$g_sy[207]$ F$g_scrape_feed$
N02160 G1 X$g_sx[208]$ Y$g_sy[208]$ F$g_scrape_feed$
N02170 G1 X$g_sx[209]$ Y$g_sy[209]$ F$g_scrape_feed$
N02180 G1 X$g_sx[210]$ Y$g_sy[210]$ F$g_scrape_feed$
N02190 G1 X$g_sx[211]$ Y$g_sy[211]$ F$g_scrape_feed$
N02200 G1 X$g_sx[212]$ Y$g_sy[212]$ F$g_scrape_feed$
N02210 G1 X$g_sx[213]$ Y$g_sy[213]$ F$g_scrape_feed$
N02220 G1 X$g_sx[214]$ Y$g_sy[214]$ F$g_scrape_feed$
N02230 G1 X$g_sx[215]$ Y$g_sy[215]$ F$g_scrape_feed$
N02240 G1 X$g_sx[216]$ Y$g_sy[216]$ F$g_scrape_feed$
N02250 G1 X$g_sx[217]$ Y$g_sy[217]$ F$g_scrape_feed$
N02260 G1 X$g_sx[218]$ Y$g_sy[218]$ F$g_scrape_feed$
N02270 G1 X$g_sx[219]$ Y$g_sy[219]$ F$g_scrape_feed$
N02280 G1 X$g_sx[220]$ Y$g_sy[220]$ F$g_scrape_feed$
N02290 G1 X$g_sx[221]$ Y$g_sy[221]$ F$g_scrape_feed$
N02300 G1 X$g_sx[222]$ Y$g_sy[222]$ F$g_scrape_feed$
N02310 G1 X$g_sx[223]$ Y$g_sy[223]$ F$g_scrape_feed$
N02320 G1 X$g_sx[224]$ Y$g_sy[224]$ F$g_scrape_feed$
N02330 G1 X$g_sx[225]$ Y$g_sy[225]$ F$g_scrape_feed$
N02340 G1 X$g_sx[226]$ Y$g_sy[226]$ F$g_scrape_feed$
N02350 G1 X$g_sx[227]$ Y$g_sy[227]$ F$g_scrape_feed$
N02360 G1 X$g_sx[228]$ Y$g_sy[228]$ F$g_scrape_feed$
N02370 G1 X$g_sx[229]$ Y$g_sy[229]$ F$g_scrape_feed$
N02380 G1 X$g_sx[230]$ Y$g_sy[230]$ F$g_scrape_feed$
N02390 G1 X$g_sx[231]$ Y$g_sy[231]$ F$g_scrape_feed$
N02400 G1 X$g_sx[232]$ Y$g_sy[232]$ F$g_scrape_feed$
N02410 G1 X$g_sx[233]$ Y$g_sy[233]$ F$g_scrape_feed$
N02420 G1 X$g_sx[234]$ Y$g_sy[234]$ F$g_scrape_feed$
N02430 G1 X$g_sx[235]$ Y$g_sy[235]$ F$g_scrape_feed$
N02440 G1 X$g_sx[236]$ Y$g_sy[236]$ F$g_scrape_feed$
N02450 G1 X$g_sx[237]$ Y$g_sy[237]$ F$g_scrape_feed$
N02460 G1 X$g_sx[238]$ Y$g_sy[238]$ F$g_scrape_feed$
N02470 G1 X$g_sx[239]$ Y$g_sy[239]$ F$g_scrape_feed$
N02480 G1 X$g_sx[240]$ Y$g_sy[240]$ F$g_scrape_feed$
N02490 G1 X$g_sx[241]$ Y$g_sy[241]$ F$g_scrape_feed$
N02500 G1 X$g_sx[242]$ Y$g_sy[242]$ F$g_scrape_feed$
N02510 G1 X$g_sx[243]$ Y$g_sy[243]$ F$g_scrape_feed$
N02520 G1 X$g_sx[244]$ Y$g_sy[244]$ F$g_scrape_feed$
N02530 G1 X$g_sx[245]$ Y$g_sy[245]$ F$g_scrape_feed$
N02540 G1 X$g_sx[246]$ Y$g_sy[246]$ F$g_scrape_feed$
N02550 G1 X$g_sx[247]$ Y$g_sy[247]$ F$g_scrape_feed$
N02560 G1 X$g_sx[248]$ Y$g_sy[248]$ F$g_scrape_feed$
N02570 G1 X$g_sx[249]$ Y$g_sy[249]$ F$g_scrape_feed$
N02580 G1 X$g_sx[250]$ Y$g_sy[250]$ F$g_scrape_feed$
N02590 G1 X$g_sx[251]$ Y$g_sy[251]$ F$g_scrape_feed$
N02600 G1 X$g_sx[252]$ Y$g_sy[252]$ F$g_scrape_feed$
N02610 G1 X$g_sx[253]$ Y$g_sy[253]$ F$g_scrape_feed$
N02620 G1 X$g_sx[254]$ Y$g_sy[254]$ F$g_scrape_feed$
N02630 G1 X$g_sx[255]$ Y$g_sy[255]$ F$g_scrape_feed$
N02640 G1 X$g_sx[256]$ Y$g_sy[256]$ F$g_scrape_feed$
N02650 G1 X$g_sx[257]$ Y$g_sy[257]$ F$g_scrape_feed$
N02660 G1 X$g_sx[258]$ Y$g_sy[258]$ F$g_scrape_feed$
N02670 G1 X$g_sx[259]$ Y$g_sy[259]$ F$g_scrape_feed$
N02680 G1 X$g_sx[260]$ Y$g_sy[260]$ F$g_scrape_feed$
N02690 G1 X$g_sx[261]$ Y$g_sy[261]$ F$g_scrape_feed$
N02700 G1 X$g_sx[262]$ Y$g_sy[262]$ F$g_scrape_feed$
N02710 G1 X$g_sx[263]$ Y$g_sy[263]$ F$g_scrape_feed$
N02720 G1 X$g_sx[264]$ Y$g_sy[264]$ F$g_scrape_feed$
N02730 G1 X$g_sx[265]$ Y$g_sy[265]$ F$g_scrape_feed$
N02740 G1 X$g_sx[266]$ Y$g_sy[266]$ F$g_scrape_feed$
N02750 G1 X$g_sx[267]$ Y$g_sy[267]$ F$g_scrape_feed$
N02760 G1 X$g_sx[268]$ Y$g_sy[268]$ F$g_scrape_feed$
N02770 G1 X$g_sx[269]$ Y$g_sy[269]$ F$g_scrape_feed$
N02780 G1 X$g_sx[270]$ Y$g_sy[270]$ F$g_scrape_feed$
N02790 G1 X$g_sx[271]$ Y$g_sy[271]$ F$g_scrape_feed$
N02800 G1 X$g_sx[272]$ Y$g_sy[272]$ F$g_scrape_feed$
N02810 G1 X$g_sx[273]$ Y$g_sy[273]$ F$g_scrape_feed$
N02820 G1 X$g_sx[274]$ Y$g_sy[274]$ F$g_scrape_feed$
N02830 G1 X$g_sx[275]$ Y$g_sy[275]$ F$g_scrape_feed$
N02840 G1 X$g_sx[276]$ Y$g_sy[276]$ F$g_scrape_feed$
N02850 G1 X$g_sx[277]$ Y$g_sy[277]$ F$g_scrape_feed$
N02860 G1 X$g_sx[278]$ Y$g_sy[278]$ F$g_scrape_feed$
N02870 G1 X$g_sx[279]$ Y$g_sy[279]$ F$g_scrape_feed$
N02880 G1 X$g_sx[280]$ Y$g_sy[280]$ F$g_scrape_feed$
N02890 G1 X$g_sx[281]$ Y$g_sy[281]$ F$g_scrape_feed$
N02900 G1 X$g_sx[282]$ Y$g_sy[282]$ F$g_scrape_feed$
N02910 G1 X$g_sx[283]$ Y$g_sy[283]$ F$g_scrape_feed$
N02920 G1 X$g_sx[284]$ Y$g_sy[284]$ F$g_scrape_feed$
N02930 G1 X$g_sx[285]$ Y$g_sy[285]$ F$g_scrape_feed$
N02940 G1 X$g_sx[286]$ Y$g_sy[286]$ F$g_scrape_feed$
N02950 G1 X$g_sx[287]$ Y$g_sy[287]$ F$g_scrape_feed$
N02960 G1 X$g_sx[288]$ Y$g_sy[288]$ F$g_scrape_feed$
N02970 G1 X$g_sx[289]$ Y$g_sy[289]$ F$g_scrape_feed$
N02980 G1 X$g_sx[290]$ Y$g_sy[290]$ F$g_scrape_feed$
N02990 G1 X$g_sx[291]$ Y$g_sy[291]$ F$g_scrape_feed$
N03000 G1 X$g_sx[292]$ Y$g_sy[292]$ F$g_scrape_feed$
N03010 G1 X$g_sx[293]$ Y$g_sy[293]$ F$g_scrape_feed$
N03020 G1 X$g_sx[294]$ Y$g_sy[294]$ F$g_scrape_feed$
N03030 G1 X$g_sx[295]$ Y$g_sy[295]$ F$g_scrape_feed$
N03040 G1 X$g_sx[296]$ Y$g_sy[296]$ F$g_scrape_feed$
N03050 G1 X$g_sx[297]$ Y$g_sy[297]$ F$g_scrape_feed$
N03060 G1 X$g_sx[298]$ Y$g_sy[298]$ F$g_scrape_feed$
N03070 G1 X$g_sx[299]$ Y$g_sy[299]$ F$g_scrape_feed$
N03080 G1 X$g_sx[300]$ Y$g_sy[300]$ F$g_scrape_feed$
N03090 G1 X$g_sx[301]$ Y$g_sy[301]$ F$g_scrape_feed$
N03100 G1 X$g_sx[302]$ Y$g_sy[302]$ F$g_scrape_feed$
N03110 G1 X$g_sx[303]$ Y$g_sy[303]$ F$g_scrape_feed$
N03120 G1 X$g_sx[304]$ Y$g_sy[304]$ F$g_scrape_feed$
N03130 G1 X$g_sx[305]$ Y$g_sy[305]$ F$g_scrape_feed$
N03140 G1 X$g_sx[306]$ Y$g_sy[306]$ F$g_scrape_feed$
N03150 G1 X$g_sx[307]$ Y$g_sy[307]$ F$g_scrape_feed$
N03160 G1 X$g_sx[308]$ Y$g_sy[308]$ F$g_scrape_feed$
N03170 G1 X$g_sx[309]$ Y$g_sy[309]$ F$g_scrape_feed$
N03180 G1 X$g_sx[310]$ Y$g_sy[310]$ F$g_scrape_feed$
N03190 G1 X$g_sx[311]$ Y$g_sy[311]$ F$g_scrape_feed$
N03200 G1 X$g_sx[312]$ Y$g_sy[312]$ F$g_scrape_feed$
N03210 G1 X$g_sx[313]$ Y$g_sy[313]$ F$g_scrape_feed$
N03220 G1 X$g_sx[314]$ Y$g_sy[314]$ F$g_scrape_feed$
N03230 G1 X$g_sx[315]$ Y$g_sy[315]$ F$g_scrape_feed$
N03240 G1 X$g_sx[316]$ Y$g_sy[316]$ F$g_scrape_feed$
N03250 G1 X$g_sx[317]$ Y$g_sy[317]$ F$g_scrape_feed$
N03260 G1 X$g_sx[318]$ Y$g_sy[318]$ F$g_scrape_feed$
N03270 G1 X$g_sx[319]$ Y$g_sy[319]$ F$g_scrape_feed$
N03280 G1 X$g_sx[320]$ Y$g_sy[320]$ F$g_scrape_feed$
N03290 G1 X$g_sx[321]$ Y$g_sy[321]$ F$g_scrape_feed$
N03300 G1 X$g_sx[322]$ Y$g_sy[322]$ F$g_scrape_feed$
N03310 G1 X$g_sx[323]$ Y$g_sy[323]$ F$g_scrape_feed$
N03320 G1 X$g_sx[324]$ Y$g_sy[324]$ F$g_scrape_feed$
N03330 G1 X$g_sx[325]$ Y$g_sy[325]$ F$g_scrape_feed$
N03340 G1 X$g_sx[326]$ Y$g_sy[326]$ F$g_scrape_feed$
N03350 G1 X$g_sx[327]$ Y$g_sy[327]$ F$g_scrape_feed$
N03360 G1 X$g_sx[328]$ Y$g_sy[328]$ F$g_scrape_feed$
N03370 G1 X$g_sx[329]$ Y$g_sy[329]$ F$g_scrape_feed$
N03380 G1 X$g_sx[330]$ Y$g_sy[330]$ F$g_scrape_feed$
N03390 G1 X$g_sx[331]$ Y$g_sy[331]$ F$g_scrape_feed$
N03400 G1 X$g_sx[332]$ Y$g_sy[332]$ F$g_scrape_feed$
N03410 G1 X$g_sx[333]$ Y$g_sy[333]$ F$g_scrape_feed$
N03420 G1 X$g_sx[334]$ Y$g_sy[334]$ F$g_scrape_feed$
N03430 G1 X$g_sx[335]$ Y$g_sy[335]$ F$g_scrape_feed$
N03440 G1 X$g_sx[336]$ Y$g_sy[336]$ F$g_scrape_feed$
N03450 G1 X$g_sx[337]$ Y$g_sy[337]$ F$g_scrape_feed$
N03460 G1 X$g_sx[338]$ Y$g_sy[338]$ F$g_scrape_feed$
N03470 G1 X$g_sx[339]$ Y$g_sy[339]$ F$g_scrape_feed$
N03480 G1 X$g_sx[340]$ Y$g_sy[340]$ F$g_scrape_feed$
N03490 G1 X$g_sx[341]$ Y$g_sy[341]$ F$g_scrape_feed$
N03500 G1 X$g_sx[342]$ Y$g_sy[342]$ F$g_scrape_feed$
N03510 G1 X$g_sx[343]$ Y$g_sy[343]$ F$g_scrape_feed$
N03520 G1 X$g_sx[344]$ Y$g_sy[344]$ F$g_scrape_feed$
N03530 G1 X$g_sx[345]$ Y$g_sy[345]$ F$g_scrape_feed$
N03540 G1 X$g_sx[346]$ Y$g_sy[346]$ F$g_scrape_feed$
N03550 G1 X$g_sx[347]$ Y$g_sy[347]$ F$g_scrape_feed$
N03560 G1 X$g_sx[348]$ Y$g_sy[348]$ F$g_scrape_feed$
N03570 G1 X$g_sx[349]$ Y$g_sy[349]$ F$g_scrape_feed$
N03580 G1 X$g_sx[350]$ Y$g_sy[350]$ F$g_scrape_feed$
N03590 G1 X$g_sx[351]$ Y$g_sy[351]$ F$g_scrape_feed$
N03600 G1 X$g_sx[352]$ Y$g_sy[352]$ F$g_scrape_feed$
N03610 G1 X$g_sx[353]$ Y$g_sy[353]$ F$g_scrape_feed$
N03620 G1 X$g_sx[354]$ Y$g_sy[354]$ F$g_scrape_feed$
N03630 G1 X$g_sx[355]$ Y$g_sy[355]$ F$g_scrape_feed$
N03640 G1 X$g_sx[356]$ Y$g_sy[356]$ F$g_scrape_feed$
N03650 G1 X$g_sx[357]$ Y$g_sy[357]$ F$g_scrape_feed$
N03660 G1 X$g_sx[358]$ Y$g_sy[358]$ F$g_scrape_feed$
N03670 G1 X$g_sx[359]$ Y$g_sy[359]$ F$g_scrape_feed$
N03680 G1 X$g_sx[360]$ Y$g_sy[360]$ F$g_scrape_feed$
N03690 G1 X$g_sx[361]$ Y$g_sy[361]$ F$g_scrape_feed$
N03700 G1 X$g_sx[362]$ Y$g_sy[362]$ F$g_scrape_feed$
N03710 G1 X$g_sx[363]$ Y$g_sy[363]$ F$g_scrape_feed$
N03720 G1 X$g_sx[364]$ Y$g_sy[364]$ F$g_scrape_feed$
N03730 G1 X$g_sx[365]$ Y$g_sy[365]$ F$g_scrape_feed$
N03740 G1 X$g_sx[366]$ Y$g_sy[366]$ F$g_scrape_feed$
N03750 G1 X$g_sx[367]$ Y$g_sy[367]$ F$g_scrape_feed$
N03760 G1 X$g_sx[368]$ Y$g_sy[368]$ F$g_scrape_feed$
N03770 G1 X$g_sx[369]$ Y$g_sy[369]$ F$g_scrape_feed$
N03780 G1 X$g_sx[370]$ Y$g_sy[370]$ F$g_scrape_feed$
N03790 G1 X$g_sx[371]$ Y$g_sy[371]$ F$g_scrape_feed$
N03800 G1 X$g_sx[372]$ Y$g_sy[372]$ F$g_scrape_feed$
N03810 G1 X$g_sx[373]$ Y$g_sy[373]$ F$g_scrape_feed$
N03820 G1 X$g_sx[374]$ Y$g_sy[374]$ F$g_scrape_feed$
N03830 G1 X$g_sx[375]$ Y$g_sy[375]$ F$g_scrape_feed$
N03840 G1 X$g_sx[376]$ Y$g_sy[376]$ F$g_scrape_feed$
N03850 G1 X$g_sx[377]$ Y$g_sy[377]$ F$g_scrape_feed$
N03860 G1 X$g_sx[378]$ Y$g_sy[378]$ F$g_scrape_feed$
N03870 G1 X$g_sx[379]$ Y$g_sy[379]$ F$g_scrape_feed$
N03880 G1 X$g_sx[380]$ Y$g_sy[380]$ F$g_scrape_feed$
N03890 G1 X$g_sx[381]$ Y$g_sy[381]$ F$g_scrape_feed$
N03900 G1 X$g_sx[382]$ Y$g_sy[382]$ F$g_scrape_feed$
N03910 G1 X$g_sx[383]$ Y$g_sy[383]$ F$g_scrape_feed$
N03920 G1 X$g_sx[384]$ Y$g_sy[384]$ F$g_scrape_feed$
N03930 G1 X$g_sx[385]$ Y$g_sy[385]$ F$g_scrape_feed$
N03940 G1 X$g_sx[386]$ Y$g_sy[386]$ F$g_scrape_feed$
N03950 G1 X$g_sx[387]$ Y$g_sy[387]$ F$g_scrape_feed$
N03960 G1 X$g_sx[388]$ Y$g_sy[388]$ F$g_scrape_feed$
N03970 G1 X$g_sx[389]$ Y$g_sy[389]$ F$g_scrape_feed$
N03980 G1 X$g_sx[390]$ Y$g_sy[390]$ F$g_scrape_feed$
N03990 G1 X$g_sx[391]$ Y$g_sy[391]$ F$g_scrape_feed$
N04000 G1 X$g_sx[392]$ Y$g_sy[392]$ F$g_scrape_feed$
N04010 G1 X$g_sx[393]$ Y$g_sy[393]$ F$g_scrape_feed$
N04020 G1 X$g_sx[394]$ Y$g_sy[394]$ F$g_scrape_feed$
N04030 G1 X$g_sx[395]$ Y$g_sy[395]$ F$g_scrape_feed$
N04040 G1 X$g_sx[396]$ Y$g_sy[396]$ F$g_scrape_feed$
N04050 G1 X$g_sx[397]$ Y$g_sy[397]$ F$g_scrape_feed$
N04060 G1 X$g_sx[398]$ Y$g_sy[398]$ F$g_scrape_feed$
N04070 G1 X$g_sx[399]$ Y$g_sy[399]$ F$g_scrape_feed$
N04080 G1 X$g_sx[400]$ Y$g_sy[400]$ F$g_scrape_feed$


N4081 M15
N4082 G0 Z 5.0

N04120 G0 X$g_cx[1]$ Y$g_cy[1]$
N04130 G1 X$g_cx[1]$ Y$g_cy[1]$ F$g_scrape_feed$
N04140 G1 X$g_cx[2]$ Y$g_cy[2]$ F$g_scrape_feed$
N04150 G1 X$g_cx[3]$ Y$g_cy[3]$ F$g_scrape_feed$
N04160 G1 X$g_cx[4]$ Y$g_cy[4]$ F$g_scrape_feed$
N04170 G1 X$g_cx[5]$ Y$g_cy[5]$ F$g_scrape_feed$
N04180 G1 X$g_cx[6]$ Y$g_cy[6]$ F$g_scrape_feed$
N04190 G1 X$g_cx[7]$ Y$g_cy[7]$ F$g_scrape_feed$
N04200 G1 X$g_cx[8]$ Y$g_cy[8]$ F$g_scrape_feed$
N04210 G1 X$g_cx[9]$ Y$g_cy[9]$ F$g_scrape_feed$
N04220 G1 X$g_cx[10]$ Y$g_cy[10]$ F$g_scrape_feed$
N04230 G1 X$g_cx[11]$ Y$g_cy[11]$ F$g_scrape_feed$
N04240 G1 X$g_cx[12]$ Y$g_cy[12]$ F$g_scrape_feed$
N04250 G1 X$g_cx[13]$ Y$g_cy[13]$ F$g_scrape_feed$
N04260 G1 X$g_cx[14]$ Y$g_cy[14]$ F$g_scrape_feed$
N04270 G1 X$g_cx[15]$ Y$g_cy[15]$ F$g_scrape_feed$
N04280 G1 X$g_cx[16]$ Y$g_cy[16]$ F$g_scrape_feed$
N04290 G1 X$g_cx[17]$ Y$g_cy[17]$ F$g_scrape_feed$
N04300 G1 X$g_cx[18]$ Y$g_cy[18]$ F$g_scrape_feed$
N04310 G1 X$g_cx[19]$ Y$g_cy[19]$ F$g_scrape_feed$
N04320 G1 X$g_cx[20]$ Y$g_cy[20]$ F$g_scrape_feed$
N04330 G1 X$g_cx[21]$ Y$g_cy[21]$ F$g_scrape_feed$
N04340 G1 X$g_cx[22]$ Y$g_cy[22]$ F$g_scrape_feed$
N04350 G1 X$g_cx[23]$ Y$g_cy[23]$ F$g_scrape_feed$
N04360 G1 X$g_cx[24]$ Y$g_cy[24]$ F$g_scrape_feed$
N04370 G1 X$g_cx[25]$ Y$g_cy[25]$ F$g_scrape_feed$
N04380 G1 X$g_cx[26]$ Y$g_cy[26]$ F$g_scrape_feed$
N04390 G1 X$g_cx[27]$ Y$g_cy[27]$ F$g_scrape_feed$
N04400 G1 X$g_cx[28]$ Y$g_cy[28]$ F$g_scrape_feed$
N04410 G1 X$g_cx[29]$ Y$g_cy[29]$ F$g_scrape_feed$
N04420 G1 X$g_cx[30]$ Y$g_cy[30]$ F$g_scrape_feed$
N04430 G1 X$g_cx[31]$ Y$g_cy[31]$ F$g_scrape_feed$
N04440 G1 X$g_cx[32]$ Y$g_cy[32]$ F$g_scrape_feed$
N04450 G1 X$g_cx[33]$ Y$g_cy[33]$ F$g_scrape_feed$
N04460 G1 X$g_cx[34]$ Y$g_cy[34]$ F$g_scrape_feed$
N04470 G1 X$g_cx[35]$ Y$g_cy[35]$ F$g_scrape_feed$
N04480 G1 X$g_cx[36]$ Y$g_cy[36]$ F$g_scrape_feed$
N04490 G1 X$g_cx[37]$ Y$g_cy[37]$ F$g_scrape_feed$
N04500 G1 X$g_cx[38]$ Y$g_cy[38]$ F$g_scrape_feed$
N04510 G1 X$g_cx[39]$ Y$g_cy[39]$ F$g_scrape_feed$
N04520 G1 X$g_cx[40]$ Y$g_cy[40]$ F$g_scrape_feed$
N04530 G1 X$g_cx[41]$ Y$g_cy[41]$ F$g_scrape_feed$
N04540 G1 X$g_cx[42]$ Y$g_cy[42]$ F$g_scrape_feed$
N04550 G1 X$g_cx[43]$ Y$g_cy[43]$ F$g_scrape_feed$
N04560 G1 X$g_cx[44]$ Y$g_cy[44]$ F$g_scrape_feed$
N04570 G1 X$g_cx[45]$ Y$g_cy[45]$ F$g_scrape_feed$
N04580 G1 X$g_cx[46]$ Y$g_cy[46]$ F$g_scrape_feed$
N04590 G1 X$g_cx[47]$ Y$g_cy[47]$ F$g_scrape_feed$
N04600 G1 X$g_cx[48]$ Y$g_cy[48]$ F$g_scrape_feed$
N04610 G1 X$g_cx[49]$ Y$g_cy[49]$ F$g_scrape_feed$
N04620 G1 X$g_cx[50]$ Y$g_cy[50]$ F$g_scrape_feed$
N04630 G1 X$g_cx[51]$ Y$g_cy[51]$ F$g_scrape_feed$
N04640 G1 X$g_cx[52]$ Y$g_cy[52]$ F$g_scrape_feed$
N04650 G1 X$g_cx[53]$ Y$g_cy[53]$ F$g_scrape_feed$
N04660 G1 X$g_cx[54]$ Y$g_cy[54]$ F$g_scrape_feed$
N04670 G1 X$g_cx[55]$ Y$g_cy[55]$ F$g_scrape_feed$
N04680 G1 X$g_cx[56]$ Y$g_cy[56]$ F$g_scrape_feed$
N04690 G1 X$g_cx[57]$ Y$g_cy[57]$ F$g_scrape_feed$
N04700 G1 X$g_cx[58]$ Y$g_cy[58]$ F$g_scrape_feed$
N04710 G1 X$g_cx[59]$ Y$g_cy[59]$ F$g_scrape_feed$
N04720 G1 X$g_cx[60]$ Y$g_cy[60]$ F$g_scrape_feed$
N04730 G1 X$g_cx[61]$ Y$g_cy[61]$ F$g_scrape_feed$
N04740 G1 X$g_cx[62]$ Y$g_cy[62]$ F$g_scrape_feed$
N04750 G1 X$g_cx[63]$ Y$g_cy[63]$ F$g_scrape_feed$
N04760 G1 X$g_cx[64]$ Y$g_cy[64]$ F$g_scrape_feed$
N04770 G1 X$g_cx[65]$ Y$g_cy[65]$ F$g_scrape_feed$
N04780 G1 X$g_cx[66]$ Y$g_cy[66]$ F$g_scrape_feed$
N04790 G1 X$g_cx[67]$ Y$g_cy[67]$ F$g_scrape_feed$
N04800 G1 X$g_cx[68]$ Y$g_cy[68]$ F$g_scrape_feed$
N04810 G1 X$g_cx[69]$ Y$g_cy[69]$ F$g_scrape_feed$
N04820 G1 X$g_cx[70]$ Y$g_cy[70]$ F$g_scrape_feed$
N04830 G1 X$g_cx[71]$ Y$g_cy[71]$ F$g_scrape_feed$
N04840 G1 X$g_cx[72]$ Y$g_cy[72]$ F$g_scrape_feed$
N04850 G1 X$g_cx[73]$ Y$g_cy[73]$ F$g_scrape_feed$
N04860 G1 X$g_cx[74]$ Y$g_cy[74]$ F$g_scrape_feed$
N04870 G1 X$g_cx[75]$ Y$g_cy[75]$ F$g_scrape_feed$
N04880 G1 X$g_cx[76]$ Y$g_cy[76]$ F$g_scrape_feed$
N04890 G1 X$g_cx[77]$ Y$g_cy[77]$ F$g_scrape_feed$
N04900 G1 X$g_cx[78]$ Y$g_cy[78]$ F$g_scrape_feed$
N04910 G1 X$g_cx[79]$ Y$g_cy[79]$ F$g_scrape_feed$
N04920 G1 X$g_cx[80]$ Y$g_cy[80]$ F$g_scrape_feed$
N04930 G1 X$g_cx[81]$ Y$g_cy[81]$ F$g_scrape_feed$
N04940 G1 X$g_cx[82]$ Y$g_cy[82]$ F$g_scrape_feed$
N04950 G1 X$g_cx[83]$ Y$g_cy[83]$ F$g_scrape_feed$
N04960 G1 X$g_cx[84]$ Y$g_cy[84]$ F$g_scrape_feed$
N04970 G1 X$g_cx[85]$ Y$g_cy[85]$ F$g_scrape_feed$
N04980 G1 X$g_cx[86]$ Y$g_cy[86]$ F$g_scrape_feed$
N04990 G1 X$g_cx[87]$ Y$g_cy[87]$ F$g_scrape_feed$
N05000 G1 X$g_cx[88]$ Y$g_cy[88]$ F$g_scrape_feed$
N05010 G1 X$g_cx[89]$ Y$g_cy[89]$ F$g_scrape_feed$
N05020 G1 X$g_cx[90]$ Y$g_cy[90]$ F$g_scrape_feed$
N05030 G1 X$g_cx[91]$ Y$g_cy[91]$ F$g_scrape_feed$
N05040 G1 X$g_cx[92]$ Y$g_cy[92]$ F$g_scrape_feed$
N05050 G1 X$g_cx[93]$ Y$g_cy[93]$ F$g_scrape_feed$
N05060 G1 X$g_cx[94]$ Y$g_cy[94]$ F$g_scrape_feed$
N05070 G1 X$g_cx[95]$ Y$g_cy[95]$ F$g_scrape_feed$
N05080 G1 X$g_cx[96]$ Y$g_cy[96]$ F$g_scrape_feed$
N05090 G1 X$g_cx[97]$ Y$g_cy[97]$ F$g_scrape_feed$
N05100 G1 X$g_cx[98]$ Y$g_cy[98]$ F$g_scrape_feed$
N05110 G1 X$g_cx[99]$ Y$g_cy[99]$ F$g_scrape_feed$
N05120 G1 X$g_cx[100]$ Y$g_cy[100]$ F$g_scrape_feed$
N05130 G1 X$g_cx[101]$ Y$g_cy[101]$ F$g_scrape_feed$
N05140 G1 X$g_cx[102]$ Y$g_cy[102]$ F$g_scrape_feed$
N05150 G1 X$g_cx[103]$ Y$g_cy[103]$ F$g_scrape_feed$
N05160 G1 X$g_cx[104]$ Y$g_cy[104]$ F$g_scrape_feed$
N05170 G1 X$g_cx[105]$ Y$g_cy[105]$ F$g_scrape_feed$
N05180 G1 X$g_cx[106]$ Y$g_cy[106]$ F$g_scrape_feed$
N05190 G1 X$g_cx[107]$ Y$g_cy[107]$ F$g_scrape_feed$
N05200 G1 X$g_cx[108]$ Y$g_cy[108]$ F$g_scrape_feed$
N05210 G1 X$g_cx[109]$ Y$g_cy[109]$ F$g_scrape_feed$
N05220 G1 X$g_cx[110]$ Y$g_cy[110]$ F$g_scrape_feed$
N05230 G1 X$g_cx[111]$ Y$g_cy[111]$ F$g_scrape_feed$
N05240 G1 X$g_cx[112]$ Y$g_cy[112]$ F$g_scrape_feed$
N05250 G1 X$g_cx[113]$ Y$g_cy[113]$ F$g_scrape_feed$
N05260 G1 X$g_cx[114]$ Y$g_cy[114]$ F$g_scrape_feed$
N05270 G1 X$g_cx[115]$ Y$g_cy[115]$ F$g_scrape_feed$
N05280 G1 X$g_cx[116]$ Y$g_cy[116]$ F$g_scrape_feed$
N05290 G1 X$g_cx[117]$ Y$g_cy[117]$ F$g_scrape_feed$
N05300 G1 X$g_cx[118]$ Y$g_cy[118]$ F$g_scrape_feed$
N05310 G1 X$g_cx[119]$ Y$g_cy[119]$ F$g_scrape_feed$
N05320 G1 X$g_cx[120]$ Y$g_cy[120]$ F$g_scrape_feed$
N05330 G1 X$g_cx[121]$ Y$g_cy[121]$ F$g_scrape_feed$
N05340 G1 X$g_cx[122]$ Y$g_cy[122]$ F$g_scrape_feed$
N05350 G1 X$g_cx[123]$ Y$g_cy[123]$ F$g_scrape_feed$
N05360 G1 X$g_cx[124]$ Y$g_cy[124]$ F$g_scrape_feed$
N05370 G1 X$g_cx[125]$ Y$g_cy[125]$ F$g_scrape_feed$
N05380 G1 X$g_cx[126]$ Y$g_cy[126]$ F$g_scrape_feed$
N05390 G1 X$g_cx[127]$ Y$g_cy[127]$ F$g_scrape_feed$
N05400 G1 X$g_cx[128]$ Y$g_cy[128]$ F$g_scrape_feed$
N05410 G1 X$g_cx[129]$ Y$g_cy[129]$ F$g_scrape_feed$
N05420 G1 X$g_cx[130]$ Y$g_cy[130]$ F$g_scrape_feed$
N05430 G1 X$g_cx[131]$ Y$g_cy[131]$ F$g_scrape_feed$
N05440 G1 X$g_cx[132]$ Y$g_cy[132]$ F$g_scrape_feed$
N05450 G1 X$g_cx[133]$ Y$g_cy[133]$ F$g_scrape_feed$
N05460 G1 X$g_cx[134]$ Y$g_cy[134]$ F$g_scrape_feed$
N05470 G1 X$g_cx[135]$ Y$g_cy[135]$ F$g_scrape_feed$
N05480 G1 X$g_cx[136]$ Y$g_cy[136]$ F$g_scrape_feed$
N05490 G1 X$g_cx[137]$ Y$g_cy[137]$ F$g_scrape_feed$
N05500 G1 X$g_cx[138]$ Y$g_cy[138]$ F$g_scrape_feed$
N05510 G1 X$g_cx[139]$ Y$g_cy[139]$ F$g_scrape_feed$
N05520 G1 X$g_cx[140]$ Y$g_cy[140]$ F$g_scrape_feed$
N05530 G1 X$g_cx[141]$ Y$g_cy[141]$ F$g_scrape_feed$
N05540 G1 X$g_cx[142]$ Y$g_cy[142]$ F$g_scrape_feed$
N05550 G1 X$g_cx[143]$ Y$g_cy[143]$ F$g_scrape_feed$
N05560 G1 X$g_cx[144]$ Y$g_cy[144]$ F$g_scrape_feed$
N05570 G1 X$g_cx[145]$ Y$g_cy[145]$ F$g_scrape_feed$
N05580 G1 X$g_cx[146]$ Y$g_cy[146]$ F$g_scrape_feed$
N05590 G1 X$g_cx[147]$ Y$g_cy[147]$ F$g_scrape_feed$
N05600 G1 X$g_cx[148]$ Y$g_cy[148]$ F$g_scrape_feed$
N05610 G1 X$g_cx[149]$ Y$g_cy[149]$ F$g_scrape_feed$
N05620 G1 X$g_cx[150]$ Y$g_cy[150]$ F$g_scrape_feed$
N05630 G1 X$g_cx[151]$ Y$g_cy[151]$ F$g_scrape_feed$
N05640 G1 X$g_cx[152]$ Y$g_cy[152]$ F$g_scrape_feed$
N05650 G1 X$g_cx[153]$ Y$g_cy[153]$ F$g_scrape_feed$
N05660 G1 X$g_cx[154]$ Y$g_cy[154]$ F$g_scrape_feed$
N05670 G1 X$g_cx[155]$ Y$g_cy[155]$ F$g_scrape_feed$
N05680 G1 X$g_cx[156]$ Y$g_cy[156]$ F$g_scrape_feed$
N05690 G1 X$g_cx[157]$ Y$g_cy[157]$ F$g_scrape_feed$
N05700 G1 X$g_cx[158]$ Y$g_cy[158]$ F$g_scrape_feed$
N05710 G1 X$g_cx[159]$ Y$g_cy[159]$ F$g_scrape_feed$
N05720 G1 X$g_cx[160]$ Y$g_cy[160]$ F$g_scrape_feed$
N05730 G1 X$g_cx[161]$ Y$g_cy[161]$ F$g_scrape_feed$
N05740 G1 X$g_cx[162]$ Y$g_cy[162]$ F$g_scrape_feed$
N05750 G1 X$g_cx[163]$ Y$g_cy[163]$ F$g_scrape_feed$
N05760 G1 X$g_cx[164]$ Y$g_cy[164]$ F$g_scrape_feed$
N05770 G1 X$g_cx[165]$ Y$g_cy[165]$ F$g_scrape_feed$
N05780 G1 X$g_cx[166]$ Y$g_cy[166]$ F$g_scrape_feed$
N05790 G1 X$g_cx[167]$ Y$g_cy[167]$ F$g_scrape_feed$
N05800 G1 X$g_cx[168]$ Y$g_cy[168]$ F$g_scrape_feed$
N05810 G1 X$g_cx[169]$ Y$g_cy[169]$ F$g_scrape_feed$
N05820 G1 X$g_cx[170]$ Y$g_cy[170]$ F$g_scrape_feed$
N05830 G1 X$g_cx[171]$ Y$g_cy[171]$ F$g_scrape_feed$
N05840 G1 X$g_cx[172]$ Y$g_cy[172]$ F$g_scrape_feed$
N05850 G1 X$g_cx[173]$ Y$g_cy[173]$ F$g_scrape_feed$
N05860 G1 X$g_cx[174]$ Y$g_cy[174]$ F$g_scrape_feed$
N05870 G1 X$g_cx[175]$ Y$g_cy[175]$ F$g_scrape_feed$
N05880 G1 X$g_cx[176]$ Y$g_cy[176]$ F$g_scrape_feed$
N05890 G1 X$g_cx[177]$ Y$g_cy[177]$ F$g_scrape_feed$
N05900 G1 X$g_cx[178]$ Y$g_cy[178]$ F$g_scrape_feed$
N05910 G1 X$g_cx[179]$ Y$g_cy[179]$ F$g_scrape_feed$
N05920 G1 X$g_cx[180]$ Y$g_cy[180]$ F$g_scrape_feed$
N05930 G1 X$g_cx[181]$ Y$g_cy[181]$ F$g_scrape_feed$
N05940 G1 X$g_cx[182]$ Y$g_cy[182]$ F$g_scrape_feed$
N05950 G1 X$g_cx[183]$ Y$g_cy[183]$ F$g_scrape_feed$
N05960 G1 X$g_cx[184]$ Y$g_cy[184]$ F$g_scrape_feed$
N05970 G1 X$g_cx[185]$ Y$g_cy[185]$ F$g_scrape_feed$
N05980 G1 X$g_cx[186]$ Y$g_cy[186]$ F$g_scrape_feed$
N05990 G1 X$g_cx[187]$ Y$g_cy[187]$ F$g_scrape_feed$
N06000 G1 X$g_cx[188]$ Y$g_cy[188]$ F$g_scrape_feed$
N06010 G1 X$g_cx[189]$ Y$g_cy[189]$ F$g_scrape_feed$
N06020 G1 X$g_cx[190]$ Y$g_cy[190]$ F$g_scrape_feed$
N06030 G1 X$g_cx[191]$ Y$g_cy[191]$ F$g_scrape_feed$
N06040 G1 X$g_cx[192]$ Y$g_cy[192]$ F$g_scrape_feed$
N06050 G1 X$g_cx[193]$ Y$g_cy[193]$ F$g_scrape_feed$
N06060 G1 X$g_cx[194]$ Y$g_cy[194]$ F$g_scrape_feed$
N06070 G1 X$g_cx[195]$ Y$g_cy[195]$ F$g_scrape_feed$
N06080 G1 X$g_cx[196]$ Y$g_cy[196]$ F$g_scrape_feed$
N06090 G1 X$g_cx[197]$ Y$g_cy[197]$ F$g_scrape_feed$
N06100 G1 X$g_cx[198]$ Y$g_cy[198]$ F$g_scrape_feed$
N06110 G1 X$g_cx[199]$ Y$g_cy[199]$ F$g_scrape_feed$
N06120 G1 X$g_cx[200]$ Y$g_cy[200]$ F$g_scrape_feed$
N06130 G1 X$g_cx[201]$ Y$g_cy[201]$ F$g_scrape_feed$
N06140 G1 X$g_cx[202]$ Y$g_cy[202]$ F$g_scrape_feed$
N06150 G1 X$g_cx[203]$ Y$g_cy[203]$ F$g_scrape_feed$
N06160 G1 X$g_cx[204]$ Y$g_cy[204]$ F$g_scrape_feed$
N06170 G1 X$g_cx[205]$ Y$g_cy[205]$ F$g_scrape_feed$
N06180 G1 X$g_cx[206]$ Y$g_cy[206]$ F$g_scrape_feed$
N06190 G1 X$g_cx[207]$ Y$g_cy[207]$ F$g_scrape_feed$
N06200 G1 X$g_cx[208]$ Y$g_cy[208]$ F$g_scrape_feed$
N06210 G1 X$g_cx[209]$ Y$g_cy[209]$ F$g_scrape_feed$
N06220 G1 X$g_cx[210]$ Y$g_cy[210]$ F$g_scrape_feed$
N06230 G1 X$g_cx[211]$ Y$g_cy[211]$ F$g_scrape_feed$
N06240 G1 X$g_cx[212]$ Y$g_cy[212]$ F$g_scrape_feed$
N06250 G1 X$g_cx[213]$ Y$g_cy[213]$ F$g_scrape_feed$
N06260 G1 X$g_cx[214]$ Y$g_cy[214]$ F$g_scrape_feed$
N06270 G1 X$g_cx[215]$ Y$g_cy[215]$ F$g_scrape_feed$
N06280 G1 X$g_cx[216]$ Y$g_cy[216]$ F$g_scrape_feed$
N06290 G1 X$g_cx[217]$ Y$g_cy[217]$ F$g_scrape_feed$
N06300 G1 X$g_cx[218]$ Y$g_cy[218]$ F$g_scrape_feed$
N06310 G1 X$g_cx[219]$ Y$g_cy[219]$ F$g_scrape_feed$
N06320 G1 X$g_cx[220]$ Y$g_cy[220]$ F$g_scrape_feed$
N06330 G1 X$g_cx[221]$ Y$g_cy[221]$ F$g_scrape_feed$
N06340 G1 X$g_cx[222]$ Y$g_cy[222]$ F$g_scrape_feed$
N06350 G1 X$g_cx[223]$ Y$g_cy[223]$ F$g_scrape_feed$
N06360 G1 X$g_cx[224]$ Y$g_cy[224]$ F$g_scrape_feed$
N06370 G1 X$g_cx[225]$ Y$g_cy[225]$ F$g_scrape_feed$
N06380 G1 X$g_cx[226]$ Y$g_cy[226]$ F$g_scrape_feed$
N06390 G1 X$g_cx[227]$ Y$g_cy[227]$ F$g_scrape_feed$
N06400 G1 X$g_cx[228]$ Y$g_cy[228]$ F$g_scrape_feed$
N06410 G1 X$g_cx[229]$ Y$g_cy[229]$ F$g_scrape_feed$
N06420 G1 X$g_cx[230]$ Y$g_cy[230]$ F$g_scrape_feed$
N06430 G1 X$g_cx[231]$ Y$g_cy[231]$ F$g_scrape_feed$
N06440 G1 X$g_cx[232]$ Y$g_cy[232]$ F$g_scrape_feed$
N06450 G1 X$g_cx[233]$ Y$g_cy[233]$ F$g_scrape_feed$
N06460 G1 X$g_cx[234]$ Y$g_cy[234]$ F$g_scrape_feed$
N06470 G1 X$g_cx[235]$ Y$g_cy[235]$ F$g_scrape_feed$
N06480 G1 X$g_cx[236]$ Y$g_cy[236]$ F$g_scrape_feed$
N06490 G1 X$g_cx[237]$ Y$g_cy[237]$ F$g_scrape_feed$
N06500 G1 X$g_cx[238]$ Y$g_cy[238]$ F$g_scrape_feed$
N06510 G1 X$g_cx[239]$ Y$g_cy[239]$ F$g_scrape_feed$
N06520 G1 X$g_cx[240]$ Y$g_cy[240]$ F$g_scrape_feed$
N06530 G1 X$g_cx[241]$ Y$g_cy[241]$ F$g_scrape_feed$
N06540 G1 X$g_cx[242]$ Y$g_cy[242]$ F$g_scrape_feed$
N06550 G1 X$g_cx[243]$ Y$g_cy[243]$ F$g_scrape_feed$
N06560 G1 X$g_cx[244]$ Y$g_cy[244]$ F$g_scrape_feed$
N06570 G1 X$g_cx[245]$ Y$g_cy[245]$ F$g_scrape_feed$
N06580 G1 X$g_cx[246]$ Y$g_cy[246]$ F$g_scrape_feed$
N06590 G1 X$g_cx[247]$ Y$g_cy[247]$ F$g_scrape_feed$
N06600 G1 X$g_cx[248]$ Y$g_cy[248]$ F$g_scrape_feed$
N06610 G1 X$g_cx[249]$ Y$g_cy[249]$ F$g_scrape_feed$
N06620 G1 X$g_cx[250]$ Y$g_cy[250]$ F$g_scrape_feed$
N06630 G1 X$g_cx[251]$ Y$g_cy[251]$ F$g_scrape_feed$
N06640 G1 X$g_cx[252]$ Y$g_cy[252]$ F$g_scrape_feed$
N06650 G1 X$g_cx[253]$ Y$g_cy[253]$ F$g_scrape_feed$
N06660 G1 X$g_cx[254]$ Y$g_cy[254]$ F$g_scrape_feed$
N06670 G1 X$g_cx[255]$ Y$g_cy[255]$ F$g_scrape_feed$
N06680 G1 X$g_cx[256]$ Y$g_cy[256]$ F$g_scrape_feed$
N06690 G1 X$g_cx[257]$ Y$g_cy[257]$ F$g_scrape_feed$
N06700 G1 X$g_cx[258]$ Y$g_cy[258]$ F$g_scrape_feed$
N06710 G1 X$g_cx[259]$ Y$g_cy[259]$ F$g_scrape_feed$
N06720 G1 X$g_cx[260]$ Y$g_cy[260]$ F$g_scrape_feed$
N06730 G1 X$g_cx[261]$ Y$g_cy[261]$ F$g_scrape_feed$
N06740 G1 X$g_cx[262]$ Y$g_cy[262]$ F$g_scrape_feed$
N06750 G1 X$g_cx[263]$ Y$g_cy[263]$ F$g_scrape_feed$
N06760 G1 X$g_cx[264]$ Y$g_cy[264]$ F$g_scrape_feed$
N06770 G1 X$g_cx[265]$ Y$g_cy[265]$ F$g_scrape_feed$
N06780 G1 X$g_cx[266]$ Y$g_cy[266]$ F$g_scrape_feed$
N06790 G1 X$g_cx[267]$ Y$g_cy[267]$ F$g_scrape_feed$
N06800 G1 X$g_cx[268]$ Y$g_cy[268]$ F$g_scrape_feed$
N06810 G1 X$g_cx[269]$ Y$g_cy[269]$ F$g_scrape_feed$
N06820 G1 X$g_cx[270]$ Y$g_cy[270]$ F$g_scrape_feed$
N06830 G1 X$g_cx[271]$ Y$g_cy[271]$ F$g_scrape_feed$
N06840 G1 X$g_cx[272]$ Y$g_cy[272]$ F$g_scrape_feed$
N06850 G1 X$g_cx[273]$ Y$g_cy[273]$ F$g_scrape_feed$
N06860 G1 X$g_cx[274]$ Y$g_cy[274]$ F$g_scrape_feed$
N06870 G1 X$g_cx[275]$ Y$g_cy[275]$ F$g_scrape_feed$
N06880 G1 X$g_cx[276]$ Y$g_cy[276]$ F$g_scrape_feed$
N06890 G1 X$g_cx[277]$ Y$g_cy[277]$ F$g_scrape_feed$
N06900 G1 X$g_cx[278]$ Y$g_cy[278]$ F$g_scrape_feed$
N06910 G1 X$g_cx[279]$ Y$g_cy[279]$ F$g_scrape_feed$
N06920 G1 X$g_cx[280]$ Y$g_cy[280]$ F$g_scrape_feed$
N06930 G1 X$g_cx[281]$ Y$g_cy[281]$ F$g_scrape_feed$
N06940 G1 X$g_cx[282]$ Y$g_cy[282]$ F$g_scrape_feed$
N06950 G1 X$g_cx[283]$ Y$g_cy[283]$ F$g_scrape_feed$
N06960 G1 X$g_cx[284]$ Y$g_cy[284]$ F$g_scrape_feed$
N06970 G1 X$g_cx[285]$ Y$g_cy[285]$ F$g_scrape_feed$
N06980 G1 X$g_cx[286]$ Y$g_cy[286]$ F$g_scrape_feed$
N06990 G1 X$g_cx[287]$ Y$g_cy[287]$ F$g_scrape_feed$
N07000 G1 X$g_cx[288]$ Y$g_cy[288]$ F$g_scrape_feed$
N07010 G1 X$g_cx[289]$ Y$g_cy[289]$ F$g_scrape_feed$
N07020 G1 X$g_cx[290]$ Y$g_cy[290]$ F$g_scrape_feed$
N07030 G1 X$g_cx[291]$ Y$g_cy[291]$ F$g_scrape_feed$
N07040 G1 X$g_cx[292]$ Y$g_cy[292]$ F$g_scrape_feed$
N07050 G1 X$g_cx[293]$ Y$g_cy[293]$ F$g_scrape_feed$
N07060 G1 X$g_cx[294]$ Y$g_cy[294]$ F$g_scrape_feed$
N07070 G1 X$g_cx[295]$ Y$g_cy[295]$ F$g_scrape_feed$
N07080 G1 X$g_cx[296]$ Y$g_cy[296]$ F$g_scrape_feed$
N07090 G1 X$g_cx[297]$ Y$g_cy[297]$ F$g_scrape_feed$
N07100 G1 X$g_cx[298]$ Y$g_cy[298]$ F$g_scrape_feed$
N07110 G1 X$g_cx[299]$ Y$g_cy[299]$ F$g_scrape_feed$
N07120 G1 X$g_cx[300]$ Y$g_cy[300]$ F$g_scrape_feed$
N07130 G1 X$g_cx[301]$ Y$g_cy[301]$ F$g_scrape_feed$
N07140 G1 X$g_cx[302]$ Y$g_cy[302]$ F$g_scrape_feed$
N07150 G1 X$g_cx[303]$ Y$g_cy[303]$ F$g_scrape_feed$
N07160 G1 X$g_cx[304]$ Y$g_cy[304]$ F$g_scrape_feed$
N07170 G1 X$g_cx[305]$ Y$g_cy[305]$ F$g_scrape_feed$
N07180 G1 X$g_cx[306]$ Y$g_cy[306]$ F$g_scrape_feed$
N07190 G1 X$g_cx[307]$ Y$g_cy[307]$ F$g_scrape_feed$
N07200 G1 X$g_cx[308]$ Y$g_cy[308]$ F$g_scrape_feed$
N07210 G1 X$g_cx[309]$ Y$g_cy[309]$ F$g_scrape_feed$
N07220 G1 X$g_cx[310]$ Y$g_cy[310]$ F$g_scrape_feed$
N07230 G1 X$g_cx[311]$ Y$g_cy[311]$ F$g_scrape_feed$
N07240 G1 X$g_cx[312]$ Y$g_cy[312]$ F$g_scrape_feed$
N07250 G1 X$g_cx[313]$ Y$g_cy[313]$ F$g_scrape_feed$
N07260 G1 X$g_cx[314]$ Y$g_cy[314]$ F$g_scrape_feed$
N07270 G1 X$g_cx[315]$ Y$g_cy[315]$ F$g_scrape_feed$
N07280 G1 X$g_cx[316]$ Y$g_cy[316]$ F$g_scrape_feed$
N07290 G1 X$g_cx[317]$ Y$g_cy[317]$ F$g_scrape_feed$
N07300 G1 X$g_cx[318]$ Y$g_cy[318]$ F$g_scrape_feed$
N07310 G1 X$g_cx[319]$ Y$g_cy[319]$ F$g_scrape_feed$
N07320 G1 X$g_cx[320]$ Y$g_cy[320]$ F$g_scrape_feed$
N07330 G1 X$g_cx[321]$ Y$g_cy[321]$ F$g_scrape_feed$
N07340 G1 X$g_cx[322]$ Y$g_cy[322]$ F$g_scrape_feed$
N07350 G1 X$g_cx[323]$ Y$g_cy[323]$ F$g_scrape_feed$
N07360 G1 X$g_cx[324]$ Y$g_cy[324]$ F$g_scrape_feed$
N07370 G1 X$g_cx[325]$ Y$g_cy[325]$ F$g_scrape_feed$
N07380 G1 X$g_cx[326]$ Y$g_cy[326]$ F$g_scrape_feed$
N07390 G1 X$g_cx[327]$ Y$g_cy[327]$ F$g_scrape_feed$
N07400 G1 X$g_cx[328]$ Y$g_cy[328]$ F$g_scrape_feed$
N07410 G1 X$g_cx[329]$ Y$g_cy[329]$ F$g_scrape_feed$
N07420 G1 X$g_cx[330]$ Y$g_cy[330]$ F$g_scrape_feed$
N07430 G1 X$g_cx[331]$ Y$g_cy[331]$ F$g_scrape_feed$
N07440 G1 X$g_cx[332]$ Y$g_cy[332]$ F$g_scrape_feed$
N07450 G1 X$g_cx[333]$ Y$g_cy[333]$ F$g_scrape_feed$
N07460 G1 X$g_cx[334]$ Y$g_cy[334]$ F$g_scrape_feed$
N07470 G1 X$g_cx[335]$ Y$g_cy[335]$ F$g_scrape_feed$
N07480 G1 X$g_cx[336]$ Y$g_cy[336]$ F$g_scrape_feed$
N07490 G1 X$g_cx[337]$ Y$g_cy[337]$ F$g_scrape_feed$
N07500 G1 X$g_cx[338]$ Y$g_cy[338]$ F$g_scrape_feed$
N07510 G1 X$g_cx[339]$ Y$g_cy[339]$ F$g_scrape_feed$
N07520 G1 X$g_cx[340]$ Y$g_cy[340]$ F$g_scrape_feed$
N07530 G1 X$g_cx[341]$ Y$g_cy[341]$ F$g_scrape_feed$
N07540 G1 X$g_cx[342]$ Y$g_cy[342]$ F$g_scrape_feed$
N07550 G1 X$g_cx[343]$ Y$g_cy[343]$ F$g_scrape_feed$
N07560 G1 X$g_cx[344]$ Y$g_cy[344]$ F$g_scrape_feed$
N07570 G1 X$g_cx[345]$ Y$g_cy[345]$ F$g_scrape_feed$
N07580 G1 X$g_cx[346]$ Y$g_cy[346]$ F$g_scrape_feed$
N07590 G1 X$g_cx[347]$ Y$g_cy[347]$ F$g_scrape_feed$
N07600 G1 X$g_cx[348]$ Y$g_cy[348]$ F$g_scrape_feed$
N07610 G1 X$g_cx[349]$ Y$g_cy[349]$ F$g_scrape_feed$
N07620 G1 X$g_cx[350]$ Y$g_cy[350]$ F$g_scrape_feed$
N07630 G1 X$g_cx[351]$ Y$g_cy[351]$ F$g_scrape_feed$
N07640 G1 X$g_cx[352]$ Y$g_cy[352]$ F$g_scrape_feed$
N07650 G1 X$g_cx[353]$ Y$g_cy[353]$ F$g_scrape_feed$
N07660 G1 X$g_cx[354]$ Y$g_cy[354]$ F$g_scrape_feed$
N07670 G1 X$g_cx[355]$ Y$g_cy[355]$ F$g_scrape_feed$
N07680 G1 X$g_cx[356]$ Y$g_cy[356]$ F$g_scrape_feed$
N07690 G1 X$g_cx[357]$ Y$g_cy[357]$ F$g_scrape_feed$
N07700 G1 X$g_cx[358]$ Y$g_cy[358]$ F$g_scrape_feed$
N07710 G1 X$g_cx[359]$ Y$g_cy[359]$ F$g_scrape_feed$
N07720 G1 X$g_cx[360]$ Y$g_cy[360]$ F$g_scrape_feed$
N07730 G1 X$g_cx[361]$ Y$g_cy[361]$ F$g_scrape_feed$
N07740 G1 X$g_cx[362]$ Y$g_cy[362]$ F$g_scrape_feed$
N07750 G1 X$g_cx[363]$ Y$g_cy[363]$ F$g_scrape_feed$
N07760 G1 X$g_cx[364]$ Y$g_cy[364]$ F$g_scrape_feed$
N07770 G1 X$g_cx[365]$ Y$g_cy[365]$ F$g_scrape_feed$
N07780 G1 X$g_cx[366]$ Y$g_cy[366]$ F$g_scrape_feed$
N07790 G1 X$g_cx[367]$ Y$g_cy[367]$ F$g_scrape_feed$
N07800 G1 X$g_cx[368]$ Y$g_cy[368]$ F$g_scrape_feed$
N07810 G1 X$g_cx[369]$ Y$g_cy[369]$ F$g_scrape_feed$
N07820 G1 X$g_cx[370]$ Y$g_cy[370]$ F$g_scrape_feed$
N07830 G1 X$g_cx[371]$ Y$g_cy[371]$ F$g_scrape_feed$
N07840 G1 X$g_cx[372]$ Y$g_cy[372]$ F$g_scrape_feed$
N07850 G1 X$g_cx[373]$ Y$g_cy[373]$ F$g_scrape_feed$
N07860 G1 X$g_cx[374]$ Y$g_cy[374]$ F$g_scrape_feed$
N07870 G1 X$g_cx[375]$ Y$g_cy[375]$ F$g_scrape_feed$
N07880 G1 X$g_cx[376]$ Y$g_cy[376]$ F$g_scrape_feed$
N07890 G1 X$g_cx[377]$ Y$g_cy[377]$ F$g_scrape_feed$
N07900 G1 X$g_cx[378]$ Y$g_cy[378]$ F$g_scrape_feed$
N07910 G1 X$g_cx[379]$ Y$g_cy[379]$ F$g_scrape_feed$
N07920 G1 X$g_cx[380]$ Y$g_cy[380]$ F$g_scrape_feed$
N07930 G1 X$g_cx[381]$ Y$g_cy[381]$ F$g_scrape_feed$
N07940 G1 X$g_cx[382]$ Y$g_cy[382]$ F$g_scrape_feed$
N07950 G1 X$g_cx[383]$ Y$g_cy[383]$ F$g_scrape_feed$
N07960 G1 X$g_cx[384]$ Y$g_cy[384]$ F$g_scrape_feed$
N07970 G1 X$g_cx[385]$ Y$g_cy[385]$ F$g_scrape_feed$
N07980 G1 X$g_cx[386]$ Y$g_cy[386]$ F$g_scrape_feed$
N07990 G1 X$g_cx[387]$ Y$g_cy[387]$ F$g_scrape_feed$
N08000 G1 X$g_cx[388]$ Y$g_cy[388]$ F$g_scrape_feed$
N08010 G1 X$g_cx[389]$ Y$g_cy[389]$ F$g_scrape_feed$
N08020 G1 X$g_cx[390]$ Y$g_cy[390]$ F$g_scrape_feed$
N08030 G1 X$g_cx[391]$ Y$g_cy[391]$ F$g_scrape_feed$
N08040 G1 X$g_cx[392]$ Y$g_cy[392]$ F$g_scrape_feed$
N08050 G1 X$g_cx[393]$ Y$g_cy[393]$ F$g_scrape_feed$
N08060 G1 X$g_cx[394]$ Y$g_cy[394]$ F$g_scrape_feed$
N08070 G1 X$g_cx[395]$ Y$g_cy[395]$ F$g_scrape_feed$
N08080 G1 X$g_cx[396]$ Y$g_cy[396]$ F$g_scrape_feed$
N08090 G1 X$g_cx[397]$ Y$g_cy[397]$ F$g_scrape_feed$
N08100 G1 X$g_cx[398]$ Y$g_cy[398]$ F$g_scrape_feed$
N08110 G1 X$g_cx[399]$ Y$g_cy[399]$ F$g_scrape_feed$
N08120 G1 X$g_cx[400]$ Y$g_cy[400]$ F$g_scrape_feed$



N08200 G1 X335 Y0 F$g_scrape_feed$

N08300 G0 Z 5.0
*)
